C09038=1044.686,246.320,-104.218,171.561,39.501,157.497
C09039=1044.679,246.071,-104.189,171.559,39.498,157.496
C09040=1044.673,245.823,-104.160,171.556,39.496,157.496
C09041=1044.666,245.575,-104.131,171.553,39.493,157.495
C09042=1044.659,245.327,-104.102,171.551,39.491,157.495
C09043=1044.653,245.078,-104.074,171.548,39.489,157.494
C09044=1044.646,244.830,-104.045,171.546,39.486,157.493
C09045=1044.640,244.582,-104.016,171.543,39.484,157.493
C09046=1044.634,244.333,-103.988,171.541,39.481,157.492
C09047=1044.627,244.085,-103.959,171.538,39.479,157.491
C09048=1044.620,243.837,-103.930,171.535,39.476,157.491
C09049=1044.613,243.589,-103.902,171.533,39.474,157.490
C09050=1044.607,243.340,-103.873,171.530,39.472,157.490
C09051=1044.601,243.092,-103.844,171.527,39.469,157.489
C09052=1044.594,242.844,-103.816,171.525,39.467,157.488
C09053=1044.588,242.595,-103.788,171.522,39.464,157.488
C09054=1044.581,242.348,-103.759,171.520,39.462,157.487
C09055=1044.575,242.099,-103.731,171.517,39.459,157.487
C09056=1044.569,241.850,-103.701,171.515,39.457,157.486
C09057=1044.562,241.602,-103.673,171.512,39.455,157.486
C09058=1044.556,241.353,-103.645,171.509,39.452,157.485
C09059=1044.549,241.106,-103.616,171.507,39.449,157.484
C09060=1044.542,240.857,-103.589,171.504,39.447,157.484
C09061=1044.536,240.609,-103.559,171.502,39.445,157.483
C09062=1044.529,240.361,-103.532,171.499,39.443,157.483
C09063=1044.523,240.112,-103.503,171.497,39.440,157.482
C09064=1044.516,239.864,-103.475,171.494,39.437,157.481
C09065=1044.509,239.616,-103.447,171.491,39.435,157.481
C09066=1044.503,239.367,-103.418,171.490,39.433,157.480
C09067=1044.496,239.119,-103.390,171.487,39.431,157.480
C09068=1044.489,238.871,-103.362,171.485,39.428,157.479
C09069=1044.483,238.622,-103.333,171.482,39.426,157.478
C09070=1044.476,238.374,-103.305,171.479,39.423,157.478
C09071=1044.469,238.125,-103.277,171.477,39.421,157.477
C09072=1044.463,237.877,-103.249,171.474,39.419,157.477
C09073=1044.456,237.629,-103.220,171.472,39.416,157.476
C09074=1044.450,237.380,-103.193,171.469,39.414,157.475
C09075=1044.444,237.132,-103.164,171.467,39.411,157.475
C09076=1044.437,236.884,-103.136,171.464,39.409,157.474
C09077=1044.430,236.635,-103.108,171.462,39.407,157.474
C09078=1044.423,236.387,-103.080,171.459,39.404,157.473
C09079=1044.417,236.139,-103.051,171.456,39.402,157.473
C09080=1044.410,235.890,-103.024,171.454,39.400,157.472
C09081=1044.404,235.642,-102.996,171.452,39.397,157.471
C09082=1044.398,235.393,-102.968,171.450,39.394,157.471
C09083=1044.390,235.109,-102.935,171.446,39.392,157.470
C09084=1044.383,234.823,-102.903,171.443,39.389,157.469
C09085=1044.375,234.539,-102.871,171.441,39.387,157.469
C09086=1044.368,234.254,-102.839,171.438,39.384,157.468
C09087=1044.361,234.006,-102.811,171.436,39.381,157.467
C09088=1044.354,233.757,-102.783,171.433,39.378,157.467
C09089=1044.348,233.509,-102.755,171.430,39.376,157.466
C09090=1044.342,233.260,-102.727,171.428,39.374,157.466
C09091=1044.335,233.012,-102.699,171.426,39.372,157.465
C09092=1044.328,232.763,-102.672,171.424,39.369,157.465
C09093=1044.322,232.515,-102.643,171.421,39.366,157.464
C09094=1044.315,232.267,-102.615,171.418,39.364,157.463
C09095=1044.309,232.018,-102.587,171.416,39.362,157.463
C09096=1044.302,231.770,-102.559,171.413,39.360,157.462
C09097=1044.296,231.522,-102.532,171.411,39.357,157.462
C09098=1044.290,231.273,-102.504,171.409,39.354,157.461
C09099=1044.283,231.025,-102.476,171.407,39.352,157.460
C09100=1044.277,230.776,-102.448,171.404,39.350,157.460
C09101=1044.270,230.528,-102.420,171.402,39.347,157.459
C09102=1044.263,230.280,-102.393,171.399,39.345,157.459
C09103=1044.256,230.031,-102.365,171.396,39.342,157.458
C09104=1044.250,229.783,-102.337,171.395,39.340,157.457
C09105=1044.243,229.534,-102.310,171.392,39.338,157.457
C09106=1044.237,229.287,-102.282,171.390,39.335,157.456
C09107=1044.231,229.038,-102.254,171.387,39.333,157.456
C09108=1044.224,228.789,-102.226,171.384,39.330,157.455
C09109=1044.218,228.541,-102.198,171.382,39.328,157.454
C09110=1044.211,228.292,-102.171,171.380,39.325,157.454
C09111=1044.204,228.044,-102.144,171.378,39.323,157.453
C09112=1044.197,227.795,-102.117,171.375,39.321,157.453
C09113=1044.191,227.547,-102.089,171.373,39.319,157.452
C09114=1044.184,227.299,-102.061,171.370,39.316,157.452
C09115=1044.178,227.051,-102.034,171.369,39.314,157.451
C09116=1044.171,226.802,-102.006,171.366,39.312,157.451
C09117=1044.164,226.554,-101.978,171.364,39.309,157.450
C09118=1044.158,226.305,-101.951,171.361,39.306,157.449
C09119=1044.151,226.056,-101.924,171.358,39.304,157.449
C09120=1044.145,225.809,-101.897,171.357,39.302,157.448
C09121=1044.138,225.560,-101.869,171.354,39.299,157.448
C09122=1044.131,225.312,-101.841,171.352,39.297,157.447
C09123=1044.125,225.063,-101.814,171.349,39.295,157.446
C09124=1044.118,224.814,-101.787,171.347,39.292,157.446
C09125=1044.111,224.566,-101.759,171.345,39.290,157.445
C09126=1044.106,224.318,-101.732,171.343,39.287,157.445
C09127=1044.099,224.069,-101.704,171.340,39.285,157.444
C09128=1044.092,223.821,-101.677,171.337,39.283,157.444
C09129=1044.085,223.573,-101.650,171.336,39.280,157.443
C09130=1044.079,223.324,-101.623,171.333,39.277,157.442
C09131=1044.072,223.076,-101.595,171.331,39.275,157.442
C09132=1044.066,222.827,-101.567,171.328,39.273,157.441
C09133=1044.059,222.578,-101.540,171.327,39.271,157.441
C09134=1044.053,222.331,-101.513,171.324,39.268,157.440
C09135=1044.046,222.082,-101.486,171.322,39.266,157.440
C09136=1044.040,221.833,-101.459,171.319,39.263,157.439
C09137=1044.033,221.585,-101.431,171.317,39.261,157.438
C09138=1044.027,221.337,-101.405,171.315,39.258,157.438
C09139=1044.019,221.044,-101.372,171.312,39.255,157.437
C09140=1044.012,220.752,-101.340,171.310,39.253,157.436
C09141=1044.003,220.459,-101.308,171.307,39.250,157.436
C09142=1043.996,220.167,-101.276,171.304,39.247,157.435
C09143=1043.990,219.918,-101.249,171.302,39.244,157.434
C09144=1043.983,219.670,-101.222,171.299,39.242,157.434
C09145=1043.976,219.421,-101.195,171.298,39.240,157.433
C09146=1043.969,219.173,-101.168,171.295,39.237,157.433
C09147=1043.963,218.925,-101.141,171.293,39.235,157.432
C09148=1043.956,218.676,-101.114,171.290,39.233,157.432
C09149=1043.950,218.428,-101.087,171.288,39.230,157.431
C09150=1043.943,218.179,-101.060,171.286,39.228,157.430
C09151=1043.936,217.930,-101.034,171.283,39.225,157.430
C09152=1043.929,217.682,-101.006,171.282,39.223,157.429
C09153=1043.924,217.433,-100.979,171.279,39.221,157.429
C09154=1043.916,217.185,-100.952,171.277,39.218,157.428
C09155=1043.910,216.936,-100.925,171.275,39.216,157.428
C09156=1043.903,216.688,-100.899,171.273,39.213,157.427
C09157=1043.897,216.440,-100.871,171.270,39.211,157.426
C09158=1043.890,216.191,-100.845,171.268,39.208,157.426
C09159=1043.884,215.943,-100.818,171.266,39.206,157.425
C09160=1043.877,215.694,-100.790,171.263,39.204,157.425
C09161=1043.870,215.445,-100.764,171.261,39.201,157.424
C09162=1043.864,215.197,-100.737,171.259,39.199,157.424
C09163=1043.857,214.949,-100.710,171.257,39.196,157.423
C09164=1043.851,214.701,-100.684,171.254,39.194,157.422
C09165=1043.844,214.452,-100.657,171.253,39.191,157.422
C09166=1043.838,214.203,-100.630,171.250,39.189,157.421
C09167=1043.829,213.866,-100.594,171.247,39.186,157.420
C09168=1043.820,213.528,-100.558,171.245,39.182,157.420
C09169=1043.811,213.191,-100.521,171.241,39.179,157.419
C09170=1043.802,212.853,-100.485,171.238,39.176,157.418
C09171=1043.796,212.606,-100.458,171.237,39.173,157.418
C09172=1043.789,212.357,-100.431,171.234,39.171,157.417
C09173=1043.782,212.108,-100.404,171.231,39.168,157.416
C09174=1043.777,211.860,-100.378,171.230,39.166,157.416
C09175=1043.769,211.611,-100.351,171.227,39.163,157.415
C09176=1043.763,211.363,-100.325,171.226,39.161,157.415
C09177=1043.757,211.114,-100.298,171.223,39.159,157.414
C09178=1043.750,210.866,-100.271,171.221,39.156,157.414
C09179=1043.743,210.617,-100.244,171.219,39.153,157.413
C09180=1043.736,210.368,-100.218,171.217,39.151,157.412
C09181=1043.730,210.120,-100.192,171.214,39.149,157.412
C09182=1043.723,209.871,-100.165,171.213,39.146,157.411
C09183=1043.717,209.623,-100.139,171.210,39.144,157.411
C09184=1043.710,209.374,-100.112,171.208,39.141,157.410
C09185=1043.704,209.126,-100.086,171.206,39.139,157.409
C09186=1043.697,208.877,-100.059,171.203,39.137,157.409
C09187=1043.690,208.629,-100.033,171.202,39.134,157.408
C09188=1043.684,208.380,-100.006,171.199,39.132,157.408
C09189=1043.677,208.132,-99.980,171.198,39.129,157.407
C09190=1043.670,207.883,-99.954,171.195,39.127,157.407
C09191=1043.665,207.660,-99.929,171.194,39.125,157.406
C09192=1043.659,207.437,-99.906,171.191,39.122,157.406
C09193=1043.653,207.214,-99.883,171.190,39.120,157.405
C09194=1043.646,206.990,-99.859,171.187,39.118,157.405
C09195=1043.641,206.767,-99.836,171.186,39.116,157.404
C09196=1043.635,206.544,-99.812,171.184,39.114,157.404
C09197=1043.628,206.321,-99.788,171.182,39.111,157.403
C09198=1043.623,206.097,-99.764,171.181,39.110,157.403
C09199=1043.597,205.046,-99.658,170.913,39.008,157.374
C09200=1043.591,204.797,-99.633,170.910,39.006,157.373
C09201=1043.585,204.548,-99.608,170.907,39.004,157.373
C09202=1043.578,204.300,-99.583,170.905,39.003,157.373
C09203=1043.572,204.051,-99.558,170.901,39.001,157.372
C09204=1043.566,203.802,-99.532,170.899,38.999,157.372
C09205=1043.560,203.554,-99.507,170.895,38.998,157.371
C09206=1043.554,203.305,-99.483,170.893,38.996,157.371
C09207=1043.548,203.056,-99.457,170.890,38.994,157.370
C09208=1043.542,202.808,-99.432,170.887,38.993,157.370
C09209=1043.536,202.559,-99.407,170.884,38.991,157.370
C09210=1043.530,202.310,-99.382,170.882,38.989,157.369
C09211=1043.524,202.062,-99.357,170.879,38.987,157.369
C09212=1043.518,201.813,-99.332,170.876,38.986,157.368
C09213=1043.512,201.565,-99.306,170.873,38.984,157.368
C09214=1043.506,201.315,-99.282,170.870,38.982,157.368
C09215=1043.499,201.067,-99.257,170.868,38.981,157.367
C09216=1043.493,200.818,-99.232,170.864,38.979,157.367
C09217=1043.487,200.570,-99.208,170.862,38.978,157.366
C09218=1043.480,200.321,-99.183,170.859,38.976,157.366
C09219=1043.474,200.072,-99.158,170.856,38.975,157.366
C09220=1043.468,199.824,-99.133,170.853,38.973,157.365
C09221=1043.462,199.574,-99.109,170.851,38.972,157.365
C09222=1043.455,199.326,-99.084,170.848,38.970,157.364
C09223=1043.449,199.077,-99.060,170.845,38.968,157.364
C09224=1043.443,198.829,-99.034,170.842,38.967,157.364
C09225=1043.437,198.580,-99.010,170.839,38.966,157.363
C09226=1043.430,198.331,-98.985,170.837,38.964,157.363
C09227=1043.424,198.082,-98.961,170.833,38.962,157.362
C09228=1043.418,197.834,-98.936,170.831,38.961,157.362
C09229=1043.411,197.585,-98.912,170.828,38.960,157.362
C09230=1043.405,197.336,-98.887,170.825,38.958,157.361
C09231=1043.399,197.087,-98.862,170.823,38.956,157.361
C09232=1043.393,196.840,-98.838,170.820,38.954,157.360
C09233=1043.387,196.590,-98.813,170.817,38.953,157.360
C09234=1043.380,196.341,-98.789,170.814,38.952,157.360
C09235=1043.374,196.093,-98.764,170.812,38.950,157.359
C09236=1043.368,195.844,-98.740,170.809,38.949,157.359
C09237=1043.362,195.596,-98.715,170.806,38.947,157.359
C09238=1043.356,195.346,-98.690,170.804,38.945,157.358
C09239=1043.350,195.098,-98.666,170.800,38.944,157.358
C09240=1043.344,194.849,-98.641,170.798,38.943,157.357
C09241=1043.337,194.600,-98.617,170.795,38.941,157.357
C09242=1043.331,194.351,-98.592,170.792,38.939,157.357
C09243=1043.325,194.104,-98.568,170.790,38.938,157.356
C09244=1043.319,193.854,-98.543,170.786,38.937,157.356
C09245=1043.312,193.605,-98.519,170.784,38.935,157.355
C09246=1043.307,193.357,-98.494,170.782,38.934,157.355
C09247=1043.301,193.108,-98.470,170.778,38.932,157.355
C09248=1043.295,192.860,-98.446,170.776,38.930,157.354
C09249=1043.289,192.610,-98.421,170.774,38.929,157.354
C09250=1043.282,192.362,-98.397,170.770,38.928,157.354
C09251=1043.277,192.113,-98.372,170.768,38.926,157.353
C09252=1043.270,191.864,-98.348,170.765,38.925,157.353
C09253=1043.264,191.615,-98.324,170.762,38.923,157.352
C09254=1043.258,191.367,-98.300,170.760,38.921,157.352
C09255=1043.252,191.118,-98.275,170.757,38.920,157.352
C09256=1043.246,190.870,-98.251,170.754,38.919,157.351
C09257=1043.240,190.621,-98.226,170.752,38.917,157.351
C09258=1043.233,190.372,-98.202,170.749,38.916,157.351
C09259=1043.228,190.123,-98.178,170.746,38.914,157.350
C09260=1043.221,189.839,-98.150,170.743,38.912,157.350
C09261=1043.214,189.554,-98.123,170.741,38.911,157.349
C09262=1043.207,189.271,-98.095,170.737,38.909,157.349
C09263=1043.201,188.985,-98.067,170.734,38.907,157.349
C09264=1043.194,188.736,-98.043,170.732,38.906,157.348
C09265=1043.189,188.488,-98.019,170.729,38.905,157.348
C09266=1043.182,188.239,-97.995,170.727,38.903,157.347
C09267=1043.176,187.991,-97.970,170.724,38.902,157.347
C09268=1043.170,187.742,-97.946,170.721,38.900,157.347
C09269=1043.165,187.493,-97.922,170.719,38.899,157.346
C09270=1043.158,187.244,-97.897,170.716,38.897,157.346
C09271=1043.153,186.996,-97.873,170.713,38.895,157.346
C09272=1043.146,186.747,-97.849,170.711,38.894,157.345
C09273=1043.141,186.498,-97.825,170.708,38.893,157.345
C09274=1043.134,186.249,-97.801,170.705,38.892,157.345
C09275=1043.129,186.001,-97.777,170.703,38.890,157.344
C09276=1043.123,185.752,-97.753,170.701,38.888,157.344
C09277=1043.117,185.503,-97.728,170.697,38.887,157.343
C09278=1043.111,185.255,-97.705,170.695,38.885,157.343
C09279=1043.104,185.005,-97.681,170.693,38.884,157.343
C09280=1043.099,184.757,-97.657,170.690,38.882,157.342
C09281=1043.092,184.508,-97.633,170.687,38.881,157.342
C09282=1043.087,184.259,-97.609,170.685,38.880,157.342
C09283=1043.081,184.010,-97.585,170.682,38.878,157.341
C09284=1043.075,183.761,-97.561,170.680,38.877,157.341
C09285=1043.069,183.513,-97.537,170.677,38.875,157.340
C09286=1043.063,183.264,-97.514,170.674,38.874,157.340
C09287=1043.056,183.015,-97.490,170.672,38.873,157.340
C09288=1043.050,182.766,-97.466,170.669,38.872,157.340
C09289=1043.044,182.517,-97.442,170.666,38.870,157.339
C09290=1043.038,182.268,-97.419,170.664,38.869,157.339
C09291=1043.031,182.019,-97.395,170.661,38.868,157.339
C09292=1043.024,181.771,-97.372,170.659,38.866,157.338
C09293=1043.018,181.522,-97.349,170.656,38.865,157.338
C09294=1043.012,181.274,-97.325,170.653,38.864,157.338
C09295=1043.005,181.025,-97.301,170.651,38.863,157.337
C09296=1043.000,180.776,-97.278,170.648,38.861,157.337
C09297=1042.993,180.527,-97.254,170.646,38.860,157.337
C09298=1042.987,180.278,-97.230,170.643,38.859,157.336
C09299=1042.981,180.030,-97.207,170.641,38.858,157.336
C09300=1042.975,179.781,-97.183,170.638,38.856,157.336
C09301=1042.969,179.532,-97.160,170.635,38.855,157.335
C09302=1042.962,179.283,-97.136,170.633,38.854,157.335
C09303=1042.957,179.034,-97.113,170.631,38.853,157.335
C09304=1042.949,178.785,-97.090,170.628,38.851,157.334
C09305=1042.943,178.537,-97.066,170.625,38.850,157.334
C09306=1042.937,178.288,-97.043,170.623,38.849,157.334
C09307=1042.931,178.039,-97.019,170.620,38.848,157.334
C09308=1042.925,177.790,-96.996,170.618,38.846,157.333
C09309=1042.918,177.541,-96.972,170.615,38.845,157.333
C09310=1042.913,177.292,-96.949,170.613,38.844,157.333
C09311=1042.907,177.044,-96.926,170.610,38.843,157.332
C09312=1042.900,176.794,-96.902,170.608,38.841,157.332
C09313=1042.894,176.546,-96.879,170.605,38.840,157.332
C09314=1042.887,176.297,-96.856,170.602,38.839,157.331
C09315=1042.881,176.049,-96.832,170.600,38.838,157.331
C09316=1042.875,175.800,-96.809,170.598,38.837,157.331
C09317=1042.869,175.550,-96.786,170.596,38.835,157.330
C09318=1042.863,175.302,-96.762,170.592,38.834,157.330
C09319=1042.857,175.053,-96.739,170.590,38.833,157.330
C09320=1042.851,174.804,-96.715,170.588,38.832,157.329
C09321=1042.845,174.555,-96.692,170.586,38.831,157.329
C09322=1042.838,174.306,-96.670,170.582,38.829,157.329
C09323=1042.832,174.057,-96.646,170.580,38.828,157.328
C09324=1042.826,173.773,-96.620,170.578,38.827,157.328
C09325=1042.818,173.488,-96.593,170.574,38.825,157.328
C09326=1042.811,173.203,-96.566,170.572,38.823,157.327
C09327=1042.805,172.918,-96.539,170.569,38.822,157.327
C09328=1042.799,172.670,-96.516,170.566,38.821,157.327
C09329=1042.792,172.420,-96.494,170.564,38.820,157.326
C09330=1042.786,172.171,-96.471,170.562,38.818,157.326
C09331=1042.780,171.923,-96.447,170.559,38.817,157.326
C09332=1042.774,171.674,-96.424,170.556,38.816,157.325
C09333=1042.768,171.425,-96.401,170.554,38.815,157.325
C09334=1042.762,171.176,-96.377,170.552,38.814,157.325
C09335=1042.756,170.928,-96.355,170.549,38.812,157.324
C09336=1042.750,170.679,-96.332,170.547,38.811,157.324
C09337=1042.743,170.429,-96.309,170.544,38.810,157.324
C09338=1042.737,170.181,-96.285,170.542,38.809,157.324
C09339=1042.732,169.932,-96.262,170.539,38.808,157.323
C09340=1042.726,169.683,-96.239,170.537,38.806,157.323
C09341=1042.720,169.434,-96.216,170.535,38.805,157.323
C09342=1042.713,169.185,-96.193,170.533,38.804,157.322
C09343=1042.707,168.937,-96.170,170.529,38.803,157.322
C09344=1042.701,168.688,-96.147,170.527,38.801,157.322
C09345=1042.696,168.439,-96.124,170.525,38.800,157.321
C09346=1042.690,168.190,-96.101,170.522,38.799,157.321
C09347=1042.683,167.941,-96.078,170.520,38.797,157.321
C09348=1042.677,167.692,-96.055,170.518,38.796,157.321
C09349=1042.671,167.443,-96.032,170.516,38.795,157.320
C09350=1042.665,167.195,-96.009,170.512,38.794,157.320
C09351=1042.660,166.946,-95.986,170.510,38.792,157.320
C09352=1042.654,166.697,-95.963,170.508,38.791,157.319
C09353=1042.647,166.448,-95.940,170.506,38.790,157.319
C09354=1042.641,166.199,-95.917,170.503,38.789,157.319
C09355=1042.635,165.950,-95.894,170.501,38.788,157.318
C09356=1042.630,165.701,-95.871,170.499,38.787,157.318
C09357=1042.624,165.452,-95.848,170.496,38.785,157.318
C09358=1042.617,165.203,-95.826,170.494,38.784,157.317
C09359=1042.612,164.955,-95.803,170.491,38.783,157.317
C09360=1042.606,164.706,-95.780,170.489,38.782,157.317
C09361=1042.600,164.457,-95.757,170.486,38.781,157.317
C09362=1042.595,164.208,-95.734,170.484,38.779,157.316
C09363=1042.588,163.959,-95.712,170.482,38.778,157.316
C09364=1042.582,163.710,-95.689,170.480,38.777,157.316
C09365=1042.577,163.461,-95.666,170.477,38.775,157.315
C09366=1042.570,163.212,-95.643,170.475,38.774,157.315
C09367=1042.565,162.963,-95.620,170.473,38.773,157.315
C09368=1042.558,162.714,-95.597,170.471,38.772,157.314
C09369=1042.552,162.466,-95.574,170.467,38.770,157.314
C09370=1042.547,162.217,-95.551,170.465,38.769,157.314
C09371=1042.541,161.968,-95.528,170.463,38.768,157.313
C09372=1042.535,161.719,-95.505,170.460,38.767,157.313
C09373=1042.529,161.470,-95.483,170.458,38.766,157.313
C09374=1042.523,161.221,-95.460,170.456,38.765,157.313
C09375=1042.517,160.972,-95.437,170.454,38.763,157.312
C09376=1042.512,160.723,-95.415,170.451,38.762,157.312
C09377=1042.505,160.474,-95.393,170.449,38.761,157.312
C09378=1042.500,160.225,-95.370,170.447,38.760,157.311
C09379=1042.494,159.977,-95.347,170.445,38.758,157.311
C09380=1042.487,159.728,-95.324,170.442,38.757,157.311
C09381=1042.481,159.479,-95.303,170.440,38.756,157.311
C09382=1042.475,159.230,-95.280,170.437,38.755,157.310
C09383=1042.469,158.981,-95.257,170.435,38.754,157.310
C09384=1042.463,158.732,-95.236,170.432,38.753,157.310
C09385=1042.457,158.483,-95.213,170.430,38.752,157.309
C09386=1042.451,158.235,-95.191,170.428,38.751,157.309
C09387=1042.445,157.986,-95.168,170.426,38.749,157.309
C09388=1042.438,157.700,-95.142,170.423,38.748,157.309
C09389=1042.431,157.414,-95.117,170.420,38.747,157.308
C09390=1042.424,157.130,-95.091,170.418,38.746,157.308
C09391=1042.417,156.844,-95.066,170.416,38.745,157.308
C09392=1042.411,156.595,-95.043,170.412,38.744,157.307
C09393=1042.404,156.346,-95.021,170.410,38.743,157.307
C09394=1042.398,156.097,-94.999,170.408,38.742,157.307
C09395=1042.392,155.848,-94.976,170.406,38.741,157.307
C09396=1042.386,155.599,-94.954,170.403,38.739,157.306
C09397=1042.380,155.350,-94.932,170.401,38.738,157.306
C09398=1042.374,155.102,-94.909,170.399,38.737,157.306
C09399=1042.368,154.852,-94.887,170.397,38.736,157.305
C09400=1042.361,154.604,-94.865,170.394,38.735,157.305
C09401=1042.356,154.354,-94.843,170.392,38.734,157.305
C09402=1042.350,154.106,-94.821,170.390,38.733,157.305
C09403=1042.343,153.856,-94.799,170.388,38.732,157.304
C09404=1042.337,153.608,-94.777,170.386,38.731,157.304
C09405=1042.331,153.358,-94.754,170.383,38.730,157.304
C09406=1042.325,153.110,-94.732,170.381,38.729,157.304
C09407=1042.319,152.861,-94.710,170.379,38.728,157.303
C09408=1042.312,152.612,-94.688,170.377,38.726,157.303
C09409=1042.307,152.364,-94.667,170.373,38.725,157.303
C09410=1042.301,152.115,-94.644,170.371,38.724,157.302
C09411=1042.295,151.865,-94.622,170.369,38.724,157.302
C09412=1042.288,151.617,-94.600,170.367,38.723,157.302
C09413=1042.282,151.368,-94.578,170.364,38.721,157.302
C09414=1042.277,151.118,-94.556,170.362,38.720,157.302
C09415=1042.270,150.870,-94.534,170.360,38.719,157.301
C09416=1042.264,150.620,-94.512,170.358,38.718,157.301
C09417=1042.258,150.372,-94.490,170.355,38.717,157.301
C09418=1042.252,150.123,-94.468,170.353,38.716,157.300
C09419=1042.246,149.873,-94.446,170.351,38.715,157.300
C09420=1042.240,149.624,-94.423,170.349,38.714,157.300
C09421=1042.234,149.376,-94.402,170.347,38.713,157.300
C09422=1042.228,149.127,-94.380,170.344,38.712,157.299
C09423=1042.222,148.878,-94.358,170.342,38.711,157.299
C09424=1042.215,148.629,-94.336,170.340,38.710,157.299
C09425=1042.209,148.380,-94.315,170.338,38.709,157.299
C09426=1042.203,148.131,-94.292,170.335,38.708,157.298
C09427=1042.197,147.882,-94.270,170.333,38.707,157.298
C09428=1042.191,147.632,-94.249,170.331,38.706,157.298
C09429=1042.186,147.384,-94.227,170.329,38.705,157.298
C09430=1042.179,147.135,-94.205,170.326,38.703,157.297
C09431=1042.173,146.886,-94.183,170.324,38.703,157.297
C09432=1042.167,146.637,-94.162,170.322,38.702,157.297
C09433=1042.161,146.388,-94.140,170.320,38.701,157.297
C09434=1042.154,146.138,-94.118,170.318,38.699,157.296
C09435=1042.148,145.890,-94.096,170.315,38.699,157.296
C09436=1042.142,145.641,-94.075,170.313,38.698,157.296
C09437=1042.136,145.392,-94.053,170.311,38.697,157.296
C09438=1042.130,145.143,-94.032,170.309,38.696,157.295
C09439=1042.124,144.894,-94.010,170.307,38.695,157.295
C09440=1042.118,144.645,-93.988,170.304,38.694,157.295
C09441=1042.111,144.396,-93.966,170.302,38.693,157.295
C09442=1042.106,144.147,-93.945,170.300,38.692,157.294
C09443=1042.099,143.899,-93.924,170.298,38.691,157.294
C09444=1042.093,143.649,-93.902,170.296,38.690,157.294
C09445=1042.087,143.400,-93.880,170.293,38.689,157.294
C09446=1042.080,143.151,-93.859,170.291,38.688,157.293
C09447=1042.074,142.902,-93.837,170.289,38.687,157.293
C09448=1042.069,142.653,-93.816,170.287,38.686,157.293
C09449=1042.062,142.404,-93.794,170.284,38.685,157.293
C09450=1042.056,142.155,-93.773,170.282,38.684,157.292
C09451=1042.050,141.906,-93.751,170.280,38.683,157.292
C09452=1042.044,141.621,-93.726,170.278,38.682,157.292
C09453=1042.036,141.335,-93.701,170.275,38.681,157.292
C09454=1042.029,141.049,-93.677,170.272,38.680,157.291
C09455=1042.022,140.764,-93.652,170.270,38.679,157.291
C09456=1042.017,140.515,-93.630,170.268,38.678,157.291
C09457=1042.010,140.266,-93.609,170.266,38.677,157.291
C09458=1042.004,140.017,-93.587,170.263,38.676,157.290
C09459=1041.997,139.768,-93.566,170.261,38.675,157.290
C09460=1041.992,139.519,-93.545,170.259,38.674,157.290
C09461=1041.986,139.270,-93.523,170.257,38.673,157.290
C09462=1041.980,139.021,-93.502,170.255,38.672,157.289
C09463=1041.974,138.771,-93.481,170.252,38.671,157.289
C09464=1041.968,138.523,-93.459,170.250,38.670,157.289
C09465=1041.961,138.274,-93.438,170.248,38.669,157.289
C09466=1041.955,138.024,-93.417,170.246,38.668,157.288
C09467=1041.949,137.775,-93.395,170.244,38.667,157.288
C09468=1041.943,137.527,-93.374,170.241,38.666,157.288
C09469=1041.936,137.278,-93.353,170.239,38.665,157.288
C09470=1041.930,137.029,-93.331,170.237,38.664,157.287
C09471=1041.924,136.779,-93.310,170.235,38.664,157.287
C09472=1041.918,136.531,-93.289,170.233,38.663,157.287
C09473=1041.912,136.281,-93.268,170.230,38.661,157.287
C09474=1041.906,136.032,-93.246,170.229,38.661,157.287
C09475=1041.900,135.784,-93.225,170.227,38.660,157.286
C09476=1041.894,135.534,-93.205,170.225,38.659,157.286
C09477=1041.887,135.285,-93.183,170.223,38.658,157.286
C09478=1041.882,135.036,-93.162,170.220,38.657,157.286
C09479=1041.875,134.788,-93.141,170.218,38.656,157.285
C09480=1041.869,134.538,-93.120,170.216,38.655,157.285
C09481=1041.864,134.289,-93.098,170.214,38.654,157.285
C09482=1041.857,134.040,-93.077,170.211,38.653,157.285
C09483=1041.851,133.791,-93.056,170.209,38.652,157.284
C09484=1041.845,133.542,-93.035,170.207,38.651,157.284
C09485=1041.838,133.293,-93.014,170.205,38.651,157.284
C09486=1041.832,133.044,-92.993,170.203,38.650,157.284
C09487=1041.827,132.795,-92.971,170.200,38.648,157.283
C09488=1041.820,132.546,-92.951,170.198,38.648,157.283
C09489=1041.814,132.297,-92.929,170.196,38.647,157.283
C09490=1041.808,132.048,-92.908,170.194,38.646,157.283
C09491=1041.802,131.799,-92.888,170.193,38.645,157.283
C09492=1041.796,131.550,-92.866,170.191,38.644,157.282
C09493=1041.790,131.301,-92.845,170.188,38.643,157.282
C09494=1041.783,131.051,-92.825,170.186,38.642,157.282
C09495=1041.778,130.803,-92.803,170.184,38.641,157.282
C09496=1041.771,130.553,-92.783,170.182,38.641,157.281
C09497=1041.764,130.305,-92.762,170.180,38.640,157.281
C09498=1041.759,130.055,-92.741,170.177,38.639,157.281
C09499=1041.752,129.807,-92.720,170.175,38.638,157.281
C09500=1041.746,129.557,-92.700,170.173,38.637,157.281
C09501=1041.740,129.309,-92.679,170.171,38.636,157.280
C09502=1041.733,129.059,-92.658,170.169,38.636,157.280
C09503=1041.727,128.810,-92.637,170.166,38.635,157.280
C09504=1041.721,128.561,-92.617,170.164,38.634,157.280
C09505=1041.714,128.312,-92.596,170.162,38.633,157.279
C09506=1041.708,128.063,-92.575,170.160,38.632,157.279
C09507=1041.702,127.814,-92.554,170.158,38.631,157.279
C09508=1041.696,127.565,-92.534,170.157,38.631,157.279
C09509=1041.690,127.316,-92.513,170.154,38.629,157.279
C09510=1041.683,127.067,-92.492,170.152,38.629,157.278
C09511=1041.677,126.818,-92.471,170.150,38.628,157.278
C09512=1041.671,126.569,-92.451,170.148,38.627,157.278
C09513=1041.665,126.319,-92.430,170.146,38.626,157.278
C09514=1041.658,126.071,-92.410,170.143,38.626,157.278
C09515=1041.653,125.821,-92.389,170.141,38.625,157.277
C09516=1041.646,125.536,-92.365,170.139,38.623,157.277
C09517=1041.638,125.249,-92.341,170.137,38.623,157.277
C09518=1041.631,124.964,-92.317,170.134,38.622,157.277
C09519=1041.624,124.678,-92.294,170.131,38.621,157.276
C09520=1041.617,124.429,-92.273,170.129,38.620,157.276
C09521=1041.611,124.179,-92.252,170.127,38.619,157.276
C09522=1041.605,123.931,-92.233,170.126,38.618,157.276
C09523=1041.599,123.682,-92.211,170.124,38.617,157.276
C09524=1041.593,123.433,-92.191,170.122,38.617,157.275
C09525=1041.587,123.183,-92.171,170.119,38.616,157.275
C09526=1041.580,122.935,-92.150,170.117,38.615,157.275
C09527=1041.574,122.685,-92.130,170.115,38.614,157.275
C09528=1041.569,122.436,-92.109,170.113,38.613,157.274
C09529=1041.562,122.187,-92.088,170.111,38.612,157.274
C09530=1041.556,121.938,-92.068,170.108,38.611,157.274
C09531=1041.550,121.689,-92.047,170.106,38.611,157.274
C09532=1041.544,121.440,-92.027,170.105,38.609,157.274
C09533=1041.537,121.191,-92.006,170.103,38.609,157.273
C09534=1041.532,120.942,-91.986,170.101,38.608,157.273
C09535=1041.525,120.692,-91.965,170.098,38.607,157.273
C09536=1041.519,120.443,-91.945,170.096,38.606,157.273
C09537=1041.514,120.195,-91.924,170.094,38.605,157.273
C09538=1041.507,119.945,-91.904,170.092,38.604,157.272
C09539=1041.501,119.697,-91.884,170.090,38.604,157.272
C09540=1041.494,119.447,-91.863,170.089,38.603,157.272
C09541=1041.489,119.199,-91.842,170.086,38.601,157.272
C09542=1041.482,118.949,-91.822,170.084,38.601,157.271
C09543=1041.476,118.700,-91.802,170.082,38.600,157.271
C09544=1041.470,118.450,-91.781,170.080,38.599,157.271
C09545=1041.464,118.202,-91.761,170.078,38.598,157.271
C09546=1041.458,117.953,-91.741,170.075,38.598,157.271
C09547=1041.451,117.704,-91.720,170.073,38.596,157.270
C09548=1041.446,117.455,-91.699,170.072,38.596,157.270
C09549=1041.440,117.205,-91.679,170.070,38.595,157.270
C09550=1041.434,116.956,-91.659,170.068,38.594,157.270
C09551=1041.428,116.707,-91.639,170.065,38.593,157.269
C09552=1041.422,116.458,-91.618,170.063,38.592,157.269
C09553=1041.416,116.209,-91.598,170.061,38.591,157.269
C09554=1041.410,115.960,-91.578,170.059,38.590,157.269
C09555=1041.404,115.710,-91.557,170.058,38.590,157.269
C09556=1041.398,115.462,-91.537,170.055,38.589,157.268
C09557=1041.391,115.213,-91.516,170.053,38.588,157.268
C09558=1041.385,114.964,-91.496,170.051,38.587,157.268
C09559=1041.380,114.715,-91.476,170.049,38.586,157.268
C09560=1041.373,114.465,-91.456,170.047,38.585,157.267
C09561=1041.367,114.216,-91.436,170.046,38.584,157.267
C09562=1041.362,113.967,-91.415,170.043,38.583,157.267
C09563=1041.355,113.718,-91.395,170.041,38.582,157.267
C09564=1041.349,113.469,-91.375,170.039,38.582,157.267
C09565=1041.343,113.220,-91.355,170.037,38.581,157.266
C09566=1041.337,112.971,-91.335,170.035,38.580,157.266
C09567=1041.331,112.722,-91.315,170.032,38.579,157.266
C09568=1041.325,112.473,-91.295,170.031,38.578,157.266
C09569=1041.318,112.224,-91.274,170.029,38.577,157.266
C09570=1041.312,111.975,-91.254,170.027,38.577,157.265
C09571=1041.306,111.725,-91.235,170.025,38.576,157.265
C09572=1041.300,111.476,-91.215,170.023,38.575,157.265
C09573=1041.294,111.227,-91.195,170.020,38.574,157.265
C09574=1041.287,110.977,-91.174,170.018,38.573,157.265
C09575=1041.281,110.729,-91.154,170.017,38.573,157.264
C09576=1041.275,110.480,-91.135,170.015,38.572,157.264
C09577=1041.269,110.230,-91.114,170.013,38.571,157.264
C09578=1041.263,109.981,-91.095,170.011,38.571,157.264
C09579=1041.257,109.732,-91.075,170.008,38.569,157.264
C09580=1041.249,109.421,-91.050,170.006,38.568,157.263
C09581=1041.241,109.110,-91.026,170.003,38.568,157.263
C09582=1041.233,108.799,-91.001,170.001,38.567,157.263
C09583=1041.226,108.489,-90.976,169.999,38.565,157.263
C09584=1041.220,108.252,-90.957,169.996,38.565,157.262
C09585=1041.213,108.015,-90.938,169.994,38.564,157.262
C09586=1041.208,107.779,-90.919,169.992,38.563,157.262
C09587=1041.202,107.542,-90.901,169.991,38.563,157.262
C09588=1041.196,107.305,-90.882,169.989,38.562,157.262
C09589=1041.189,107.068,-90.863,169.987,38.561,157.261
C09590=1041.184,106.832,-90.844,169.984,38.561,157.261
C09591=1041.178,106.595,-90.826,169.983,38.560,157.261
C09592=1041.172,106.346,-90.806,169.981,38.559,157.261
C09593=1041.166,106.097,-90.786,169.979,38.558,157.261
C09594=1041.160,105.848,-90.766,169.977,38.558,157.261
C09595=1041.153,105.598,-90.746,169.975,38.557,157.260
C09596=1041.147,105.349,-90.726,169.973,38.556,157.260
C09597=1041.141,105.101,-90.707,169.971,38.555,157.260
C09598=1041.134,104.851,-90.688,169.969,38.554,157.260
C09599=1041.128,104.602,-90.668,169.967,38.554,157.260
C09600=1041.122,104.353,-90.648,169.965,38.553,157.259
C09601=1041.117,104.104,-90.628,169.963,38.552,157.259
C09602=1041.111,103.855,-90.608,169.960,38.551,157.259
C09603=1041.104,103.605,-90.589,169.959,38.550,157.259
C09604=1041.098,103.356,-90.569,169.957,38.550,157.259
C09605=1041.092,103.107,-90.549,169.955,38.549,157.258
C09606=1041.086,102.858,-90.530,169.953,38.548,157.258
C09607=1041.079,102.608,-90.510,169.951,38.547,157.258
C09608=1041.073,102.359,-90.491,169.948,38.546,157.258
C09609=1041.067,102.110,-90.471,169.947,38.546,157.258
C09610=1041.061,101.862,-90.451,169.945,38.545,157.257
C09611=1041.055,101.612,-90.432,169.943,38.544,157.257
C09612=1041.049,101.363,-90.412,169.941,38.543,157.257
C09613=1041.042,101.114,-90.393,169.939,38.543,157.257
C09614=1041.036,100.865,-90.373,169.936,38.541,157.257
C09615=1041.030,100.615,-90.354,169.935,38.541,157.256
C09616=1041.024,100.366,-90.334,169.933,38.540,157.256
C09617=1041.017,100.117,-90.315,169.931,38.539,157.256
C09618=1041.011,99.868,-90.295,169.929,38.539,157.256
C09619=1041.005,99.619,-90.276,169.927,38.538,157.256
C09620=1040.999,99.370,-90.256,169.924,38.537,157.255
C09621=1040.993,99.120,-90.237,169.923,38.536,157.255
C09622=1040.986,98.871,-90.217,169.921,38.536,157.255
C09623=1040.980,98.622,-90.198,169.919,38.535,157.255
C09624=1040.974,98.373,-90.179,169.917,38.534,157.255
C09625=1040.968,98.124,-90.160,169.915,38.534,157.255
C09626=1040.961,97.875,-90.141,169.913,38.533,157.254
C09627=1040.955,97.625,-90.121,169.911,38.532,157.254
C09628=1040.948,97.376,-90.102,169.909,38.531,157.254
C09629=1040.943,97.127,-90.083,169.907,38.531,157.254
C09630=1040.936,96.878,-90.063,169.905,38.530,157.254
C09631=1040.930,96.629,-90.044,169.903,38.529,157.253
C09632=1040.924,96.380,-90.025,169.901,38.529,157.253
C09633=1040.917,96.130,-90.005,169.899,38.527,157.253
C09634=1040.912,95.881,-89.986,169.897,38.527,157.253
C09635=1040.905,95.632,-89.967,169.895,38.526,157.253
C09636=1040.899,95.383,-89.947,169.893,38.525,157.252
C09637=1040.893,95.134,-89.929,169.891,38.525,157.252
C09638=1040.887,94.884,-89.909,169.889,38.524,157.252
C09639=1040.880,94.636,-89.890,169.887,38.523,157.252
C09640=1040.875,94.386,-89.871,169.885,38.522,157.252
C09641=1040.868,94.136,-89.852,169.883,38.522,157.252
C09642=1040.862,93.888,-89.832,169.881,38.521,157.251
C09643=1040.855,93.639,-89.813,169.879,38.520,157.251
C09644=1040.848,93.352,-89.791,169.877,38.520,157.251
C09645=1040.841,93.066,-89.769,169.874,38.518,157.251
C09646=1040.835,92.781,-89.747,169.872,38.518,157.251
C09647=1040.827,92.495,-89.725,169.870,38.517,157.250
C09648=1040.821,92.246,-89.706,169.868,38.516,157.250
C09649=1040.815,91.996,-89.687,169.866,38.515,157.250
C09650=1040.808,91.746,-89.668,169.864,38.515,157.250
C09651=1040.802,91.498,-89.648,169.863,38.514,157.250
C09652=1040.796,91.249,-89.629,169.860,38.513,157.249
C09653=1040.790,90.999,-89.610,169.858,38.512,157.249
C09654=1040.784,90.750,-89.592,169.856,38.512,157.249
C09655=1040.778,90.501,-89.572,169.854,38.511,157.249
C09656=1040.772,90.251,-89.554,169.853,38.510,157.249
C09657=1040.766,90.003,-89.534,169.851,38.509,157.248
C09658=1040.759,89.754,-89.515,169.848,38.508,157.248
C09659=1040.753,89.504,-89.496,169.846,38.508,157.248
C09660=1040.746,89.255,-89.478,169.844,38.507,157.248
C09661=1040.741,89.006,-89.458,169.842,38.507,157.248
C09662=1040.734,88.757,-89.440,169.841,38.506,157.247
C09663=1040.728,88.508,-89.421,169.839,38.505,157.247
C09664=1040.721,88.258,-89.402,169.837,38.504,157.247
C09665=1040.715,88.008,-89.383,169.834,38.504,157.247
C09666=1040.709,87.759,-89.364,169.832,38.503,157.247
C09667=1040.702,87.510,-89.346,169.830,38.502,157.247
C09668=1040.696,87.261,-89.327,169.829,38.502,157.246
C09669=1040.690,87.012,-89.308,169.827,38.501,157.246
C09670=1040.684,86.762,-89.289,169.825,38.501,157.246
C09671=1040.677,86.513,-89.270,169.822,38.499,157.246
C09672=1040.671,86.264,-89.252,169.820,38.499,157.246
C09673=1040.664,86.015,-89.233,169.818,38.498,157.246
C09674=1040.659,85.766,-89.214,169.817,38.498,157.245
C09675=1040.652,85.516,-89.195,169.815,38.497,157.245
C09676=1040.646,85.267,-89.177,169.813,38.496,157.245
C09677=1040.639,85.018,-89.158,169.811,38.496,157.245
C09678=1040.633,84.769,-89.139,169.808,38.495,157.245
C09679=1040.627,84.520,-89.120,169.807,38.494,157.245
C09680=1040.621,84.271,-89.101,169.805,38.493,157.244
C09681=1040.615,84.021,-89.083,169.803,38.493,157.244
C09682=1040.608,83.772,-89.064,169.801,38.492,157.244
C09683=1040.602,83.523,-89.045,169.799,38.492,157.244
C09684=1040.596,83.274,-89.026,169.797,38.491,157.244
C09685=1040.590,83.025,-89.008,169.795,38.490,157.243
C09686=1040.583,82.775,-88.990,169.793,38.489,157.243
C09687=1040.577,82.526,-88.971,169.791,38.488,157.243
C09688=1040.571,82.276,-88.952,169.789,38.488,157.243
C09689=1040.565,82.027,-88.933,169.787,38.487,157.243
C09690=1040.558,81.778,-88.914,169.786,38.487,157.243
C09691=1040.552,81.529,-88.896,169.783,38.485,157.242
C09692=1040.546,81.281,-88.878,169.781,38.485,157.242
C09693=1040.540,81.031,-88.860,169.779,38.484,157.242
C09694=1040.534,80.781,-88.840,169.777,38.484,157.242
C09695=1040.528,80.532,-88.822,169.775,38.483,157.242
C09696=1040.522,80.283,-88.803,169.774,38.482,157.242
C09697=1040.515,80.034,-88.784,169.772,38.482,157.241
C09698=1040.509,79.785,-88.766,169.769,38.480,157.241
C09699=1040.503,79.535,-88.747,169.767,38.480,157.241
C09700=1040.497,79.286,-88.729,169.765,38.479,157.241
C09701=1040.490,79.037,-88.710,169.764,38.479,157.241
C09702=1040.485,78.788,-88.692,169.762,38.478,157.240
C09703=1040.479,78.538,-88.674,169.760,38.477,157.240
C09704=1040.472,78.289,-88.655,169.758,38.477,157.240
C09705=1040.466,78.040,-88.636,169.755,38.476,157.240
C09706=1040.459,77.791,-88.618,169.754,38.475,157.240
C09707=1040.453,77.541,-88.600,169.752,38.474,157.240
C09708=1040.446,77.255,-88.578,169.750,38.474,157.239
C09709=1040.439,76.969,-88.557,169.748,38.473,157.239
C09710=1040.432,76.683,-88.536,169.746,38.472,157.239
C09711=1040.424,76.397,-88.514,169.742,38.472,157.239
C09712=1040.418,76.147,-88.496,169.741,38.470,157.239
C09713=1040.413,75.899,-88.478,169.739,38.470,157.238
C09714=1040.406,75.649,-88.461,169.737,38.469,157.238
C09715=1040.399,75.400,-88.442,169.735,38.469,157.238
C09716=1040.393,75.151,-88.423,169.733,38.468,157.238
C09717=1040.387,74.901,-88.406,169.731,38.468,157.238
C09718=1040.380,74.652,-88.387,169.729,38.466,157.238
C09719=1040.374,74.403,-88.369,169.727,38.466,157.237
C09720=1040.368,74.153,-88.350,169.725,38.465,157.237
C09721=1040.362,73.905,-88.332,169.723,38.465,157.237
C09722=1040.356,73.655,-88.314,169.721,38.464,157.237
C09723=1040.349,73.406,-88.295,169.719,38.463,157.237
C09724=1040.343,73.156,-88.277,169.718,38.463,157.237
C09725=1040.337,72.907,-88.259,169.715,38.462,157.236
C09726=1040.330,72.658,-88.241,169.713,38.461,157.236
C09727=1040.324,72.410,-88.223,169.711,38.461,157.236
C09728=1040.318,72.160,-88.205,169.709,38.460,157.236
C09729=1040.312,71.911,-88.187,169.708,38.459,157.236
C09730=1040.305,71.662,-88.168,169.706,38.459,157.236
C09731=1040.299,71.412,-88.150,169.704,38.458,157.235
C09732=1040.293,71.163,-88.132,169.702,38.458,157.235
C09733=1040.287,70.914,-88.114,169.699,38.457,157.235
C09734=1040.280,70.664,-88.096,169.697,38.456,157.235
C09735=1040.274,70.415,-88.078,169.696,38.455,157.235
C09736=1040.268,70.165,-88.060,169.694,38.455,157.235
C09737=1040.262,69.917,-88.042,169.692,38.454,157.234
C09738=1040.256,69.667,-88.024,169.690,38.454,157.234
C09739=1040.249,69.418,-88.005,169.687,38.453,157.234
C09740=1040.243,69.168,-87.987,169.686,38.452,157.234
C09741=1040.236,68.919,-87.969,169.684,38.451,157.234
C09742=1040.230,68.670,-87.951,169.682,38.451,157.234
C09743=1040.224,68.421,-87.934,169.680,38.450,157.233
C09744=1040.218,68.172,-87.915,169.678,38.450,157.233
C09745=1040.211,67.922,-87.898,169.676,38.449,157.233
C09746=1040.205,67.672,-87.880,169.675,38.448,157.233
C09747=1040.199,67.424,-87.861,169.672,38.447,157.233
C09748=1040.193,67.174,-87.843,169.670,38.447,157.233
C09749=1040.186,66.925,-87.826,169.668,38.446,157.232
C09750=1040.180,66.676,-87.807,169.666,38.446,157.232
C09751=1040.174,66.427,-87.790,169.664,38.445,157.232
C09752=1040.167,66.177,-87.773,169.663,38.444,157.232
C09753=1040.161,65.928,-87.754,169.661,38.444,157.232
C09754=1040.155,65.678,-87.736,169.658,38.443,157.232
C09755=1040.149,65.430,-87.719,169.656,38.443,157.231
C09756=1040.142,65.181,-87.700,169.654,38.442,157.231
C09757=1040.136,64.931,-87.682,169.652,38.441,157.231
C09758=1040.129,64.681,-87.665,169.651,38.441,157.231
C09759=1040.124,64.432,-87.647,169.649,38.440,157.231
C09760=1040.117,64.183,-87.629,169.647,38.439,157.231
C09761=1040.110,63.934,-87.612,169.644,38.439,157.230
C09762=1040.104,63.684,-87.594,169.642,38.438,157.230
C09763=1040.098,63.435,-87.577,169.640,38.438,157.230
C09764=1040.092,63.186,-87.559,169.639,38.437,157.230
C09765=1040.085,62.936,-87.541,169.637,38.436,157.230
C09766=1040.079,62.687,-87.523,169.635,38.436,157.230
C09767=1040.072,62.438,-87.506,169.633,38.435,157.230
C09768=1040.065,62.189,-87.488,169.631,38.435,157.229
C09769=1040.059,61.939,-87.470,169.629,38.434,157.229
C09770=1040.052,61.690,-87.453,169.626,38.434,157.229
C09771=1040.047,61.441,-87.436,169.624,38.433,157.229
C09772=1040.039,61.154,-87.415,169.622,38.433,157.229
C09773=1040.032,60.868,-87.396,169.620,38.432,157.229
C09774=1040.024,60.582,-87.376,169.618,38.432,157.229
C09775=1040.017,60.296,-87.356,169.616,38.431,157.228
C09776=1040.011,60.047,-87.337,169.614,38.431,157.228
C09777=1040.004,59.797,-87.320,169.612,38.430,157.228
C09778=1039.998,59.547,-87.302,169.609,38.429,157.228
C09779=1039.991,59.299,-87.285,169.607,38.428,157.228
C09780=1039.985,59.049,-87.267,169.606,38.428,157.228
C09781=1039.979,58.800,-87.249,169.604,38.427,157.227
C09782=1039.972,58.551,-87.232,169.602,38.427,157.227
C09783=1039.965,58.301,-87.215,169.600,38.426,157.227
C09784=1039.959,58.052,-87.197,169.598,38.426,157.227
C09785=1039.953,57.803,-87.180,169.595,38.425,157.227
C09786=1039.947,57.553,-87.162,169.593,38.424,157.227
C09787=1039.940,57.304,-87.145,169.592,38.424,157.227
C09788=1039.934,57.055,-87.128,169.590,38.423,157.226
C09789=1039.928,56.805,-87.110,169.588,38.423,157.226
C09790=1039.921,56.556,-87.093,169.586,38.422,157.226
C09791=1039.915,56.307,-87.076,169.584,38.422,157.226
C09792=1039.908,56.057,-87.058,169.582,38.421,157.226
C09793=1039.902,55.809,-87.041,169.580,38.421,157.226
C09794=1039.896,55.559,-87.023,169.578,38.420,157.226
C09795=1039.889,55.310,-87.006,169.576,38.420,157.225
C09796=1039.883,55.060,-86.989,169.574,38.419,157.225
C09797=1039.877,54.810,-86.971,169.572,38.418,157.225
C09798=1039.871,54.562,-86.954,169.570,38.418,157.225
C09799=1039.864,54.312,-86.937,169.568,38.417,157.225
C09800=1039.858,54.063,-86.919,169.566,38.417,157.225
C09801=1039.852,53.814,-86.902,169.565,38.416,157.225
C09802=1039.845,53.564,-86.885,169.562,38.415,157.224
C09803=1039.839,53.315,-86.867,169.560,38.415,157.224
C09804=1039.832,53.066,-86.850,169.558,38.414,157.224
C09805=1039.827,52.816,-86.833,169.556,38.413,157.224
C09806=1039.820,52.567,-86.816,169.554,38.413,157.224
C09807=1039.813,52.317,-86.798,169.552,38.412,157.224
C09808=1039.808,52.068,-86.781,169.551,38.412,157.223
C09809=1039.801,51.819,-86.763,169.549,38.411,157.223
C09810=1039.795,51.570,-86.746,169.546,38.411,157.223
C09811=1039.789,51.320,-86.729,169.544,38.410,157.223
C09812=1039.783,51.071,-86.712,169.542,38.410,157.223
C09813=1039.776,50.822,-86.695,169.540,38.409,157.223
C09814=1039.770,50.573,-86.677,169.539,38.409,157.223
C09815=1039.764,50.323,-86.660,169.537,38.407,157.222
C09816=1039.758,50.074,-86.644,169.535,38.407,157.222
C09817=1039.751,49.824,-86.626,169.532,38.406,157.222
C09818=1039.745,49.575,-86.609,169.530,38.406,157.222
C09819=1039.738,49.326,-86.592,169.528,38.405,157.222
C09820=1039.733,49.077,-86.574,169.526,38.405,157.222
C09821=1039.726,48.827,-86.557,169.525,38.404,157.221
C09822=1039.720,48.578,-86.540,169.523,38.403,157.221
C09823=1039.714,48.328,-86.522,169.521,38.403,157.221
C09824=1039.708,48.079,-86.506,169.519,38.402,157.221
C09825=1039.701,47.830,-86.489,169.516,38.401,157.221
C09826=1039.696,47.581,-86.471,169.514,38.401,157.221
C09827=1039.689,47.331,-86.454,169.512,38.400,157.220
C09828=1039.683,47.082,-86.438,169.511,38.400,157.220
C09829=1039.676,46.832,-86.420,169.509,38.399,157.220
C09830=1039.670,46.583,-86.403,169.507,38.398,157.220
C09831=1039.664,46.333,-86.386,169.505,38.398,157.220
C09832=1039.658,46.085,-86.369,169.503,38.397,157.220
C09833=1039.652,45.835,-86.352,169.500,38.397,157.220
C09834=1039.646,45.585,-86.335,169.499,38.396,157.219
C09835=1039.639,45.337,-86.318,169.497,38.395,157.219
C09836=1039.632,45.049,-86.298,169.495,38.395,157.219
C09837=1039.625,44.764,-86.278,169.492,38.394,157.219
C09838=1039.618,44.477,-86.259,169.490,38.393,157.219
C09839=1039.611,44.190,-86.240,169.488,38.392,157.218
C09840=1039.605,43.941,-86.223,169.485,38.392,157.218
C09841=1039.598,43.692,-86.205,169.484,38.391,157.218
C09842=1039.593,43.442,-86.188,169.482,38.391,157.218
C09843=1039.587,43.193,-86.172,169.480,38.390,157.218
C09844=1039.580,42.943,-86.155,169.478,38.390,157.218
C09845=1039.574,42.694,-86.138,169.476,38.389,157.218
C09846=1039.567,42.444,-86.121,169.474,38.388,157.217
C09847=1039.561,42.196,-86.104,169.472,38.388,157.217
C09848=1039.554,41.946,-86.088,169.469,38.387,157.217
C09849=1039.548,41.697,-86.071,169.468,38.387,157.217
C09850=1039.542,41.447,-86.054,169.466,38.386,157.217
C09851=1039.535,41.198,-86.037,169.464,38.386,157.217
C09852=1039.529,40.949,-86.021,169.462,38.385,157.217
C09853=1039.522,40.699,-86.004,169.460,38.385,157.216
C09854=1039.517,40.450,-85.987,169.458,38.384,157.216
C09855=1039.511,40.200,-85.970,169.456,38.384,157.216
C09856=1039.504,39.951,-85.953,169.454,38.383,157.216
C09857=1039.499,39.701,-85.937,169.451,38.382,157.216
C09858=1039.492,39.452,-85.920,169.450,38.381,157.216
C09859=1039.486,39.203,-85.903,169.448,38.381,157.215
C09860=1039.479,38.954,-85.886,169.446,38.380,157.215
C09861=1039.473,38.704,-85.870,169.444,38.380,157.215
C09862=1039.467,38.455,-85.853,169.442,38.379,157.215
C09863=1039.461,38.206,-85.836,169.440,38.379,157.215
C09864=1039.454,37.956,-85.820,169.437,38.378,157.215
C09865=1039.448,37.706,-85.804,169.435,38.377,157.215
C09866=1039.442,37.458,-85.787,169.433,38.377,157.214
C09867=1039.435,37.208,-85.770,169.432,38.376,157.214
C09868=1039.429,36.958,-85.754,169.430,38.376,157.214
C09869=1039.422,36.710,-85.737,169.428,38.376,157.214
C09870=1039.416,36.460,-85.721,169.426,38.375,157.214
C09871=1039.410,36.210,-85.704,169.424,38.375,157.214
C09872=1039.403,35.960,-85.688,169.422,38.374,157.214
C09873=1039.397,35.712,-85.671,169.420,38.374,157.214
C09874=1039.391,35.462,-85.655,169.417,38.373,157.213
C09875=1039.384,35.213,-85.639,169.415,38.373,157.213
C09876=1039.378,34.963,-85.622,169.413,38.372,157.213
C09877=1039.372,34.715,-85.605,169.411,38.372,157.213
C09878=1039.365,34.464,-85.589,169.410,38.371,157.213
C09879=1039.359,34.215,-85.572,169.408,38.370,157.213
C09880=1039.352,33.966,-85.557,169.406,38.370,157.213
C09881=1039.346,33.717,-85.539,169.404,38.370,157.212
C09882=1039.340,33.467,-85.523,169.402,38.369,157.212
C09883=1039.334,33.218,-85.507,169.399,38.369,157.212
C09884=1039.328,32.969,-85.491,169.397,38.368,157.212
C09885=1039.320,32.719,-85.475,169.395,38.368,157.212
C09886=1039.315,32.470,-85.458,169.393,38.367,157.212
C09887=1039.308,32.221,-85.441,169.391,38.367,157.212
C09888=1039.302,31.971,-85.425,169.389,38.366,157.211
C09889=1039.295,31.722,-85.409,169.387,38.366,157.211
C09890=1039.289,31.472,-85.393,169.385,38.365,157.211
C09891=1039.283,31.223,-85.377,169.383,38.364,157.211
C09892=1039.277,30.973,-85.360,169.381,38.364,157.211
C09893=1039.271,30.724,-85.344,169.379,38.363,157.211
C09894=1039.264,30.475,-85.327,169.377,38.363,157.211
C09895=1039.258,30.226,-85.311,169.375,38.363,157.211
C09896=1039.251,29.976,-85.294,169.373,38.362,157.210
C09897=1039.245,29.726,-85.278,169.371,38.362,157.210
C09898=1039.238,29.477,-85.263,169.369,38.361,157.210
C09899=1039.233,29.228,-85.246,169.367,38.361,157.210
C09900=1039.225,28.941,-85.227,169.365,38.360,157.210
C09901=1039.218,28.654,-85.209,169.362,38.360,157.210
C09902=1039.211,28.368,-85.190,169.360,38.358,157.209
C09903=1039.203,28.081,-85.172,169.357,38.358,157.209
C09904=1039.197,27.832,-85.155,169.355,38.358,157.209
C09905=1039.190,27.582,-85.139,169.353,38.358,157.209
C09906=1039.184,27.333,-85.123,169.352,38.357,157.209
C09907=1039.178,27.084,-85.107,169.350,38.356,157.209
C09908=1039.172,26.834,-85.092,169.348,38.356,157.209
C09909=1039.166,26.585,-85.076,169.345,38.355,157.209
C09910=1039.159,26.335,-85.059,169.343,38.355,157.208
C09911=1039.153,26.086,-85.043,169.341,38.355,157.208
C09912=1039.147,25.836,-85.027,169.339,38.354,157.208
C09913=1039.140,25.587,-85.011,169.337,38.354,157.208
C09914=1039.133,25.337,-84.995,169.335,38.353,157.208
C09915=1039.127,25.088,-84.979,169.333,38.353,157.208
C09916=1039.121,24.839,-84.963,169.331,38.352,157.208
C09917=1039.114,24.590,-84.947,169.329,38.352,157.208
C09918=1039.108,24.340,-84.931,169.327,38.352,157.208
C09919=1039.103,24.090,-84.915,169.324,38.351,157.207
C09920=1039.095,23.841,-84.899,169.322,38.351,157.207
C09921=1039.089,23.591,-84.883,169.320,38.350,157.207
C09922=1039.083,23.342,-84.867,169.318,38.349,157.207
C09923=1039.077,23.093,-84.851,169.316,38.349,157.207
C09924=1039.070,22.844,-84.835,169.314,38.349,157.207
C09925=1039.064,22.595,-84.819,169.312,38.348,157.207
C09926=1039.057,22.344,-84.804,169.310,38.348,157.206
C09927=1039.051,22.095,-84.788,169.308,38.347,157.206
C09928=1039.044,21.846,-84.772,169.307,38.347,157.206
C09929=1039.038,21.596,-84.756,169.304,38.346,157.206
C09930=1039.032,21.347,-84.740,169.302,38.346,157.206
C09931=1039.026,21.097,-84.724,169.300,38.345,157.206
C09932=1039.019,20.848,-84.709,169.298,38.345,157.206
C09933=1039.013,20.599,-84.693,169.296,38.345,157.206
C09934=1039.007,20.350,-84.677,169.294,38.344,157.205
C09935=1039.001,20.099,-84.661,169.292,38.344,157.205
C09936=1038.994,19.850,-84.645,169.290,38.343,157.205
C09937=1038.988,19.601,-84.629,169.288,38.342,157.205
C09938=1038.981,19.352,-84.613,169.286,38.343,157.205
C09939=1038.976,19.102,-84.598,169.283,38.342,157.205
C09940=1038.969,18.853,-84.582,169.281,38.342,157.205
C09941=1038.962,18.604,-84.567,169.279,38.341,157.205
C09942=1038.957,18.354,-84.551,169.277,38.340,157.204
C09943=1038.950,18.105,-84.535,169.275,38.341,157.204
C09944=1038.944,17.856,-84.519,169.273,38.340,157.204
C09945=1038.937,17.605,-84.504,169.271,38.339,157.204
C09946=1038.930,17.356,-84.488,169.269,38.339,157.204
C09947=1038.924,17.107,-84.472,169.267,38.338,157.204
C09948=1038.918,16.857,-84.457,169.265,38.338,157.204
C09949=1038.911,16.608,-84.441,169.262,38.338,157.204
C09950=1038.906,16.358,-84.426,169.260,38.337,157.203
C09951=1038.899,16.109,-84.410,169.258,38.337,157.203
C09952=1038.893,15.860,-84.394,169.256,38.336,157.203
C09953=1038.887,15.610,-84.379,169.254,38.336,157.203
C09954=1038.880,15.361,-84.363,169.252,38.336,157.203
C09955=1038.874,15.111,-84.348,169.250,38.335,157.203
C09956=1038.868,14.862,-84.332,169.248,38.335,157.203
C09957=1038.861,14.612,-84.317,169.246,38.334,157.203
C09958=1038.855,14.363,-84.301,169.244,38.334,157.202
C09959=1038.848,14.114,-84.285,169.242,38.334,157.202
C09960=1038.842,13.864,-84.270,169.239,38.333,157.202
C09961=1038.836,13.615,-84.255,169.237,38.333,157.202
C09962=1038.830,13.365,-84.239,169.235,38.332,157.202
C09963=1038.823,13.116,-84.224,169.233,38.332,157.202
C09964=1038.816,12.830,-84.206,169.231,38.332,157.202
C09965=1038.808,12.545,-84.189,169.228,38.331,157.202
C09966=1038.801,12.260,-84.171,169.226,38.331,157.202
C09967=1038.794,11.974,-84.154,169.224,38.331,157.202
C09968=1038.787,11.725,-84.138,169.222,38.330,157.201
C09969=1038.780,11.475,-84.123,169.220,38.330,157.201
C09970=1038.774,11.226,-84.108,169.218,38.330,157.201
C09971=1038.768,10.976,-84.092,169.215,38.329,157.201
C09972=1038.762,10.727,-84.077,169.213,38.329,157.201
C09973=1038.755,10.478,-84.062,169.210,38.329,157.201
C09974=1038.749,10.228,-84.047,169.208,38.328,157.201
C09975=1038.742,9.979,-84.031,169.206,38.328,157.201
C09976=1038.736,9.729,-84.016,169.204,38.328,157.201
C09977=1038.729,9.480,-84.001,169.202,38.327,157.200
C09978=1038.723,9.231,-83.985,169.200,38.327,157.200
C09979=1038.716,8.981,-83.971,169.198,38.327,157.200
C09980=1038.710,8.731,-83.956,169.196,38.326,157.200
C09981=1038.704,8.482,-83.939,169.194,38.326,157.200
C09982=1038.697,8.232,-83.924,169.191,38.325,157.200
C09983=1038.691,7.983,-83.909,169.189,38.325,157.200
C09984=1038.684,7.734,-83.894,169.187,38.325,157.200
C09985=1038.678,7.484,-83.879,169.185,38.324,157.200
C09986=1038.672,7.234,-83.864,169.183,38.324,157.199
C09987=1038.665,6.985,-83.849,169.181,38.324,157.199
C09988=1038.659,6.736,-83.833,169.179,38.323,157.199
C09989=1038.652,6.486,-83.818,169.177,38.323,157.199
C09990=1038.646,6.237,-83.804,169.175,38.323,157.199
C09991=1038.640,5.987,-83.789,169.173,38.322,157.199
C09992=1038.633,5.738,-83.773,169.171,38.321,157.199
C09993=1038.627,5.489,-83.758,169.169,38.322,157.199
C09994=1038.621,5.239,-83.743,169.166,38.321,157.199
C09995=1038.615,4.989,-83.728,169.163,38.320,157.198
C09996=1038.608,4.739,-83.713,169.161,38.321,157.198
//INST
///DATE 2021/06/17 10:57
///ATTR SC,RW,RJ
////FRAME ROBOT
///GROUP1 RB1
NOP
MOVL C00000 V=800.0 PL=0
MOVL C00001 V=800.0 PL=0
MOVL C00002 V=800.0 PL=0
MOVL C00003 V=800.0 PL=0
MOVL C00004 V=800.0 PL=0
MOVL C00005 V=800.0 PL=0
MOVL C00006 V=800.0 PL=0
MOVL C00007 V=800.0 PL=0
MOVL C00008 V=800.0 PL=0
MOVL C00009 V=800.0 PL=0
MOVL C00010 V=800.0 PL=0
MOVL C00011 V=800.0 PL=0
MOVL C00012 V=800.0 PL=0
MOVL C00013 V=800.0 PL=0
MOVL C00014 V=800.0 PL=0
MOVL C00015 V=800.0 PL=0
MOVL C00016 V=800.0 PL=0
MOVL C00017 V=800.0 PL=0
MOVL C00018 V=800.0 PL=0
MOVL C00019 V=800.0 PL=0
MOVL C00020 V=800.0 PL=0
MOVL C00021 V=800.0 PL=0
MOVL C00022 V=800.0 PL=0
MOVL C00023 V=800.0 PL=0
MOVL C00024 V=800.0 PL=0
MOVL C00025 V=800.0 PL=0
MOVL C00026 V=800.0 PL=0
MOVL C00027 V=800.0 PL=0
MOVL C00028 V=800.0 PL=0
MOVL C00029 V=800.0 PL=0
MOVL C00030 V=800.0 PL=0
MOVL C00031 V=800.0 PL=0
MOVL C00032 V=800.0 PL=0
MOVL C00033 V=800.0 PL=0
MOVL C00034 V=800.0 PL=0
MOVL C00035 V=800.0 PL=0
MOVL C00036 V=800.0 PL=0
MOVL C00037 V=800.0 PL=0
MOVL C00038 V=800.0 PL=0
MOVL C00039 V=800.0 PL=0
MOVL C00040 V=800.0 PL=0
MOVL C00041 V=800.0 PL=0
MOVL C00042 V=800.0 PL=0
MOVL C00043 V=800.0 PL=0
MOVL C00044 V=800.0 PL=0
MOVL C00045 V=800.0 PL=0
MOVL C00046 V=800.0 PL=0
MOVL C00047 V=800.0 PL=0
MOVL C00048 V=800.0 PL=0
MOVL C00049 V=800.0 PL=0
MOVL C00050 V=800.0 PL=0
MOVL C00051 V=800.0 PL=0
MOVL C00052 V=800.0 PL=0
MOVL C00053 V=800.0 PL=0
MOVL C00054 V=800.0 PL=0
MOVL C00055 V=800.0 PL=0
MOVL C00056 V=800.0 PL=0
MOVL C00057 V=800.0 PL=0
MOVL C00058 V=800.0 PL=0
MOVL C00059 V=800.0 PL=0
MOVL C00060 V=800.0 PL=0
MOVL C00061 V=800.0 PL=0
MOVL C00062 V=800.0 PL=0
MOVL C00063 V=800.0 PL=0
MOVL C00064 V=800.0 PL=0
MOVL C00065 V=800.0 PL=0
MOVL C00066 V=800.0 PL=0
MOVL C00067 V=800.0 PL=0
MOVL C00068 V=800.0 PL=0
MOVL C00069 V=800.0 PL=0
MOVL C00070 V=800.0 PL=0
MOVL C00071 V=800.0 PL=0
MOVL C00072 V=800.0 PL=0
MOVL C00073 V=800.0 PL=0
MOVL C00074 V=800.0 PL=0
MOVL C00075 V=800.0 PL=0
MOVL C00076 V=800.0 PL=0
MOVL C00077 V=800.0 PL=0
MOVL C00078 V=800.0 PL=0
MOVL C00079 V=800.0 PL=0
MOVL C00080 V=800.0 PL=0
MOVL C00081 V=800.0 PL=0
MOVL C00082 V=800.0 PL=0
MOVL C00083 V=800.0 PL=0
MOVL C00084 V=800.0 PL=0
MOVL C00085 V=800.0 PL=0
MOVL C00086 V=800.0 PL=0
MOVL C00087 V=800.0 PL=0
MOVL C00088 V=800.0 PL=0
MOVL C00089 V=800.0 PL=0
MOVL C00090 V=800.0 PL=0
MOVL C00091 V=800.0 PL=0
MOVL C00092 V=800.0 PL=0
MOVL C00093 V=800.0 PL=0
MOVL C00094 V=800.0 PL=0
MOVL C00095 V=800.0 PL=0
MOVL C00096 V=800.0 PL=0
MOVL C00097 V=800.0 PL=0
MOVL C00098 V=800.0 PL=0
MOVL C00099 V=800.0 PL=0
MOVL C00100 V=800.0 PL=0
MOVL C00101 V=800.0 PL=0
MOVL C00102 V=800.0 PL=0
MOVL C00103 V=800.0 PL=0
MOVL C00104 V=800.0 PL=0
MOVL C00105 V=800.0 PL=0
MOVL C00106 V=800.0 PL=0
MOVL C00107 V=800.0 PL=0
MOVL C00108 V=800.0 PL=0
MOVL C00109 V=800.0 PL=0
MOVL C00110 V=800.0 PL=0
MOVL C00111 V=800.0 PL=0
MOVL C00112 V=800.0 PL=0
MOVL C00113 V=800.0 PL=0
MOVL C00114 V=800.0 PL=0
MOVL C00115 V=800.0 PL=0
MOVL C00116 V=800.0 PL=0
MOVL C00117 V=800.0 PL=0
MOVL C00118 V=800.0 PL=0
MOVL C00119 V=800.0 PL=0
MOVL C00120 V=800.0 PL=0
MOVL C00121 V=800.0 PL=0
MOVL C00122 V=800.0 PL=0
MOVL C00123 V=800.0 PL=0
MOVL C00124 V=800.0 PL=0
MOVL C00125 V=800.0 PL=0
MOVL C00126 V=800.0 PL=0
MOVL C00127 V=800.0 PL=0
MOVL C00128 V=800.0 PL=0
MOVL C00129 V=800.0 PL=0
MOVL C00130 V=800.0 PL=0
MOVL C00131 V=800.0 PL=0
MOVL C00132 V=800.0 PL=0
MOVL C00133 V=800.0 PL=0
MOVL C00134 V=800.0 PL=0
MOVL C00135 V=800.0 PL=0
MOVL C00136 V=800.0 PL=0
MOVL C00137 V=800.0 PL=0
MOVL C00138 V=800.0 PL=0
MOVL C00139 V=800.0 PL=0
MOVL C00140 V=800.0 PL=0
MOVL C00141 V=800.0 PL=0
MOVL C00142 V=800.0 PL=0
MOVL C00143 V=800.0 PL=0
MOVL C00144 V=800.0 PL=0
MOVL C00145 V=800.0 PL=0
MOVL C00146 V=800.0 PL=0
MOVL C00147 V=800.0 PL=0
MOVL C00148 V=800.0 PL=0
MOVL C00149 V=800.0 PL=0
MOVL C00150 V=800.0 PL=0
MOVL C00151 V=800.0 PL=0
MOVL C00152 V=800.0 PL=0
MOVL C00153 V=800.0 PL=0
MOVL C00154 V=800.0 PL=0
MOVL C00155 V=800.0 PL=0
MOVL C00156 V=800.0 PL=0
MOVL C00157 V=800.0 PL=0
MOVL C00158 V=800.0 PL=0
MOVL C00159 V=800.0 PL=0
MOVL C00160 V=800.0 PL=0
MOVL C00161 V=800.0 PL=0
MOVL C00162 V=800.0 PL=0
MOVL C00163 V=800.0 PL=0
MOVL C00164 V=800.0 PL=0
MOVL C00165 V=800.0 PL=0
MOVL C00166 V=800.0 PL=0
MOVL C00167 V=800.0 PL=0
MOVL C00168 V=800.0 PL=0
MOVL C00169 V=800.0 PL=0
MOVL C00170 V=800.0 PL=0
MOVL C00171 V=800.0 PL=0
MOVL C00172 V=800.0 PL=0
MOVL C00173 V=800.0 PL=0
MOVL C00174 V=800.0 PL=0
MOVL C00175 V=800.0 PL=0
MOVL C00176 V=800.0 PL=0
MOVL C00177 V=800.0 PL=0
MOVL C00178 V=800.0 PL=0
MOVL C00179 V=800.0 PL=0
MOVL C00180 V=800.0 PL=0
MOVL C00181 V=800.0 PL=0
MOVL C00182 V=800.0 PL=0
MOVL C00183 V=800.0 PL=0
MOVL C00184 V=800.0 PL=0
MOVL C00185 V=800.0 PL=0
MOVL C00186 V=800.0 PL=0
MOVL C00187 V=800.0 PL=0
MOVL C00188 V=800.0 PL=0
MOVL C00189 V=800.0 PL=0
MOVL C00190 V=800.0 PL=0
MOVL C00191 V=800.0 PL=0
MOVL C00192 V=800.0 PL=0
MOVL C00193 V=800.0 PL=0
MOVL C00194 V=800.0 PL=0
MOVL C00195 V=800.0 PL=0
MOVL C00196 V=800.0 PL=0
MOVL C00197 V=800.0 PL=0
MOVL C00198 V=800.0 PL=0
MOVL C00199 V=800.0 PL=0
MOVL C00200 V=800.0 PL=0
MOVL C00201 V=800.0 PL=0
MOVL C00202 V=800.0 PL=0
MOVL C00203 V=800.0 PL=0
MOVL C00204 V=800.0 PL=0
MOVL C00205 V=800.0 PL=0
MOVL C00206 V=800.0 PL=0
MOVL C00207 V=800.0 PL=0
MOVL C00208 V=800.0 PL=0
MOVL C00209 V=800.0 PL=0
MOVL C00210 V=800.0 PL=0
MOVL C00211 V=800.0 PL=0
MOVL C00212 V=800.0 PL=0
MOVL C00213 V=800.0 PL=0
MOVL C00214 V=800.0 PL=0
MOVL C00215 V=800.0 PL=0
MOVL C00216 V=800.0 PL=0
MOVL C00217 V=800.0 PL=0
MOVL C00218 V=800.0 PL=0
MOVL C00219 V=800.0 PL=0
MOVL C00220 V=800.0 PL=0
MOVL C00221 V=800.0 PL=0
MOVL C00222 V=800.0 PL=0
MOVL C00223 V=800.0 PL=0
MOVL C00224 V=800.0 PL=0
MOVL C00225 V=800.0 PL=0
MOVL C00226 V=800.0 PL=0
MOVL C00227 V=800.0 PL=0
MOVL C00228 V=800.0 PL=0
MOVL C00229 V=800.0 PL=0
MOVL C00230 V=800.0 PL=0
MOVL C00231 V=800.0 PL=0
MOVL C00232 V=800.0 PL=0
MOVL C00233 V=800.0 PL=0
MOVL C00234 V=800.0 PL=0
MOVL C00235 V=800.0 PL=0
MOVL C00236 V=800.0 PL=0
MOVL C00237 V=800.0 PL=0
MOVL C00238 V=800.0 PL=0
MOVL C00239 V=800.0 PL=0
MOVL C00240 V=800.0 PL=0
MOVL C00241 V=800.0 PL=0
MOVL C00242 V=800.0 PL=0
MOVL C00243 V=800.0 PL=0
MOVL C00244 V=800.0 PL=0
MOVL C00245 V=800.0 PL=0
MOVL C00246 V=800.0 PL=0
MOVL C00247 V=800.0 PL=0
MOVL C00248 V=800.0 PL=0
MOVL C00249 V=800.0 PL=0
MOVL C00250 V=800.0 PL=0
MOVL C00251 V=800.0 PL=0
MOVL C00252 V=800.0 PL=0
MOVL C00253 V=800.0 PL=0
MOVL C00254 V=800.0 PL=0
MOVL C00255 V=800.0 PL=0
MOVL C00256 V=800.0 PL=0
MOVL C00257 V=800.0 PL=0
MOVL C00258 V=800.0 PL=0
MOVL C00259 V=800.0 PL=0
MOVL C00260 V=800.0 PL=0
MOVL C00261 V=800.0 PL=0
MOVL C00262 V=800.0 PL=0
MOVL C00263 V=800.0 PL=0
MOVL C00264 V=800.0 PL=0
MOVL C00265 V=800.0 PL=0
MOVL C00266 V=800.0 PL=0
MOVL C00267 V=800.0 PL=0
MOVL C00268 V=800.0 PL=0
MOVL C00269 V=800.0 PL=0
MOVL C00270 V=800.0 PL=0
MOVL C00271 V=800.0 PL=0
MOVL C00272 V=800.0 PL=0
MOVL C00273 V=800.0 PL=0
MOVL C00274 V=800.0 PL=0
MOVL C00275 V=800.0 PL=0
MOVL C00276 V=800.0 PL=0
MOVL C00277 V=800.0 PL=0
MOVL C00278 V=800.0 PL=0
MOVL C00279 V=800.0 PL=0
MOVL C00280 V=800.0 PL=0
MOVL C00281 V=800.0 PL=0
MOVL C00282 V=800.0 PL=0
MOVL C00283 V=800.0 PL=0
MOVL C00284 V=800.0 PL=0
MOVL C00285 V=800.0 PL=0
MOVL C00286 V=800.0 PL=0
MOVL C00287 V=800.0 PL=0
MOVL C00288 V=800.0 PL=0
MOVL C00289 V=800.0 PL=0
MOVL C00290 V=800.0 PL=0
MOVL C00291 V=800.0 PL=0
MOVL C00292 V=800.0 PL=0
MOVL C00293 V=800.0 PL=0
MOVL C00294 V=800.0 PL=0
MOVL C00295 V=800.0 PL=0
MOVL C00296 V=800.0 PL=0
MOVL C00297 V=800.0 PL=0
MOVL C00298 V=800.0 PL=0
MOVL C00299 V=800.0 PL=0
MOVL C00300 V=800.0 PL=0
MOVL C00301 V=800.0 PL=0
MOVL C00302 V=800.0 PL=0
MOVL C00303 V=800.0 PL=0
MOVL C00304 V=800.0 PL=0
MOVL C00305 V=800.0 PL=0
MOVL C00306 V=800.0 PL=0
MOVL C00307 V=800.0 PL=0
MOVL C00308 V=800.0 PL=0
MOVL C00309 V=800.0 PL=0
MOVL C00310 V=800.0 PL=0
MOVL C00311 V=800.0 PL=0
MOVL C00312 V=800.0 PL=0
MOVL C00313 V=800.0 PL=0
MOVL C00314 V=800.0 PL=0
MOVL C00315 V=800.0 PL=0
MOVL C00316 V=800.0 PL=0
MOVL C00317 V=800.0 PL=0
MOVL C00318 V=800.0 PL=0
MOVL C00319 V=800.0 PL=0
MOVL C00320 V=800.0 PL=0
MOVL C00321 V=800.0 PL=0
MOVL C00322 V=800.0 PL=0
MOVL C00323 V=800.0 PL=0
MOVL C00324 V=800.0 PL=0
MOVL C00325 V=800.0 PL=0
MOVL C00326 V=800.0 PL=0
MOVL C00327 V=800.0 PL=0
MOVL C00328 V=800.0 PL=0
MOVL C00329 V=800.0 PL=0
MOVL C00330 V=800.0 PL=0
MOVL C00331 V=800.0 PL=0
MOVL C00332 V=800.0 PL=0
MOVL C00333 V=800.0 PL=0
MOVL C00334 V=800.0 PL=0
MOVL C00335 V=800.0 PL=0
MOVL C00336 V=800.0 PL=0
MOVL C00337 V=800.0 PL=0
MOVL C00338 V=800.0 PL=0
MOVL C00339 V=800.0 PL=0
MOVL C00340 V=800.0 PL=0
MOVL C00341 V=800.0 PL=0
MOVL C00342 V=800.0 PL=0
MOVL C00343 V=800.0 PL=0
MOVL C00344 V=800.0 PL=0
MOVL C00345 V=800.0 PL=0
MOVL C00346 V=800.0 PL=0
MOVL C00347 V=800.0 PL=0
MOVL C00348 V=800.0 PL=0
MOVL C00349 V=800.0 PL=0
MOVL C00350 V=800.0 PL=0
MOVL C00351 V=800.0 PL=0
MOVL C00352 V=800.0 PL=0
MOVL C00353 V=800.0 PL=0
MOVL C00354 V=800.0 PL=0
MOVL C00355 V=800.0 PL=0
MOVL C00356 V=800.0 PL=0
MOVL C00357 V=800.0 PL=0
MOVL C00358 V=800.0 PL=0
MOVL C00359 V=800.0 PL=0
MOVL C00360 V=800.0 PL=0
MOVL C00361 V=800.0 PL=0
MOVL C00362 V=800.0 PL=0
MOVL C00363 V=800.0 PL=0
MOVL C00364 V=800.0 PL=0
MOVL C00365 V=800.0 PL=0
MOVL C00366 V=800.0 PL=0
MOVL C00367 V=800.0 PL=0
MOVL C00368 V=800.0 PL=0
MOVL C00369 V=800.0 PL=0
MOVL C00370 V=800.0 PL=0
MOVL C00371 V=800.0 PL=0
MOVL C00372 V=800.0 PL=0
MOVL C00373 V=800.0 PL=0
MOVL C00374 V=800.0 PL=0
MOVL C00375 V=800.0 PL=0
MOVL C00376 V=800.0 PL=0
MOVL C00377 V=800.0 PL=0
MOVL C00378 V=800.0 PL=0
MOVL C00379 V=800.0 PL=0
MOVL C00380 V=800.0 PL=0
MOVL C00381 V=800.0 PL=0
MOVL C00382 V=800.0 PL=0
MOVL C00383 V=800.0 PL=0
MOVL C00384 V=800.0 PL=0
MOVL C00385 V=800.0 PL=0
MOVL C00386 V=800.0 PL=0
MOVL C00387 V=800.0 PL=0
MOVL C00388 V=800.0 PL=0
MOVL C00389 V=800.0 PL=0
MOVL C00390 V=800.0 PL=0
MOVL C00391 V=800.0 PL=0
MOVL C00392 V=800.0 PL=0
MOVL C00393 V=800.0 PL=0
MOVL C00394 V=800.0 PL=0
MOVL C00395 V=800.0 PL=0
MOVL C00396 V=800.0 PL=0
MOVL C00397 V=800.0 PL=0
MOVL C00398 V=800.0 PL=0
MOVL C00399 V=800.0 PL=0
MOVL C00400 V=800.0 PL=0
MOVL C00401 V=800.0 PL=0
MOVL C00402 V=800.0 PL=0
MOVL C00403 V=800.0 PL=0
MOVL C00404 V=800.0 PL=0
MOVL C00405 V=800.0 PL=0
MOVL C00406 V=800.0 PL=0
MOVL C00407 V=800.0 PL=0
MOVL C00408 V=800.0 PL=0
MOVL C00409 V=800.0 PL=0
MOVL C00410 V=800.0 PL=0
MOVL C00411 V=800.0 PL=0
MOVL C00412 V=800.0 PL=0
MOVL C00413 V=800.0 PL=0
MOVL C00414 V=800.0 PL=0
MOVL C00415 V=800.0 PL=0
MOVL C00416 V=800.0 PL=0
MOVL C00417 V=800.0 PL=0
MOVL C00418 V=800.0 PL=0
MOVL C00419 V=800.0 PL=0
MOVL C00420 V=800.0 PL=0
MOVL C00421 V=800.0 PL=0
MOVL C00422 V=800.0 PL=0
MOVL C00423 V=800.0 PL=0
MOVL C00424 V=800.0 PL=0
MOVL C00425 V=800.0 PL=0
MOVL C00426 V=800.0 PL=0
MOVL C00427 V=800.0 PL=0
MOVL C00428 V=800.0 PL=0
MOVL C00429 V=800.0 PL=0
MOVL C00430 V=800.0 PL=0
MOVL C00431 V=800.0 PL=0
MOVL C00432 V=800.0 PL=0
MOVL C00433 V=800.0 PL=0
MOVL C00434 V=800.0 PL=0
MOVL C00435 V=800.0 PL=0
MOVL C00436 V=800.0 PL=0
MOVL C00437 V=800.0 PL=0
MOVL C00438 V=800.0 PL=0
MOVL C00439 V=800.0 PL=0
MOVL C00440 V=800.0 PL=0
MOVL C00441 V=800.0 PL=0
MOVL C00442 V=800.0 PL=0
MOVL C00443 V=800.0 PL=0
MOVL C00444 V=800.0 PL=0
MOVL C00445 V=800.0 PL=0
MOVL C00446 V=800.0 PL=0
MOVL C00447 V=800.0 PL=0
MOVL C00448 V=800.0 PL=0
MOVL C00449 V=800.0 PL=0
MOVL C00450 V=800.0 PL=0
MOVL C00451 V=800.0 PL=0
MOVL C00452 V=800.0 PL=0
MOVL C00453 V=800.0 PL=0
MOVL C00454 V=800.0 PL=0
MOVL C00455 V=800.0 PL=0
MOVL C00456 V=800.0 PL=0
MOVL C00457 V=800.0 PL=0
MOVL C00458 V=800.0 PL=0
MOVL C00459 V=800.0 PL=0
MOVL C00460 V=800.0 PL=0
MOVL C00461 V=800.0 PL=0
MOVL C00462 V=800.0 PL=0
MOVL C00463 V=800.0 PL=0
MOVL C00464 V=800.0 PL=0
MOVL C00465 V=800.0 PL=0
MOVL C00466 V=800.0 PL=0
MOVL C00467 V=800.0 PL=0
MOVL C00468 V=800.0 PL=0
MOVL C00469 V=800.0 PL=0
MOVL C00470 V=800.0 PL=0
MOVL C00471 V=800.0 PL=0
MOVL C00472 V=800.0 PL=0
MOVL C00473 V=800.0 PL=0
MOVL C00474 V=800.0 PL=0
MOVL C00475 V=800.0 PL=0
MOVL C00476 V=800.0 PL=0
MOVL C00477 V=800.0 PL=0
MOVL C00478 V=800.0 PL=0
MOVL C00479 V=800.0 PL=0
MOVL C00480 V=800.0 PL=0
MOVL C00481 V=800.0 PL=0
MOVL C00482 V=800.0 PL=0
MOVL C00483 V=800.0 PL=0
MOVL C00484 V=800.0 PL=0
MOVL C00485 V=800.0 PL=0
MOVL C00486 V=800.0 PL=0
MOVL C00487 V=800.0 PL=0
MOVL C00488 V=800.0 PL=0
MOVL C00489 V=800.0 PL=0
MOVL C00490 V=800.0 PL=0
MOVL C00491 V=800.0 PL=0
MOVL C00492 V=800.0 PL=0
MOVL C00493 V=800.0 PL=0
MOVL C00494 V=800.0 PL=0
MOVL C00495 V=800.0 PL=0
MOVL C00496 V=800.0 PL=0
MOVL C00497 V=800.0 PL=0
MOVL C00498 V=800.0 PL=0
MOVL C00499 V=800.0 PL=0
MOVL C00500 V=800.0 PL=0
MOVL C00501 V=800.0 PL=0
MOVL C00502 V=800.0 PL=0
MOVL C00503 V=800.0 PL=0
MOVL C00504 V=800.0 PL=0
MOVL C00505 V=800.0 PL=0
MOVL C00506 V=800.0 PL=0
MOVL C00507 V=800.0 PL=0
MOVL C00508 V=800.0 PL=0
MOVL C00509 V=800.0 PL=0
MOVL C00510 V=800.0 PL=0
MOVL C00511 V=800.0 PL=0
MOVL C00512 V=800.0 PL=0
MOVL C00513 V=800.0 PL=0
MOVL C00514 V=800.0 PL=0
MOVL C00515 V=800.0 PL=0
MOVL C00516 V=800.0 PL=0
MOVL C00517 V=800.0 PL=0
MOVL C00518 V=800.0 PL=0
MOVL C00519 V=800.0 PL=0
MOVL C00520 V=800.0 PL=0
MOVL C00521 V=800.0 PL=0
MOVL C00522 V=800.0 PL=0
MOVL C00523 V=800.0 PL=0
MOVL C00524 V=800.0 PL=0
MOVL C00525 V=800.0 PL=0
MOVL C00526 V=800.0 PL=0
MOVL C00527 V=800.0 PL=0
MOVL C00528 V=800.0 PL=0
MOVL C00529 V=800.0 PL=0
MOVL C00530 V=800.0 PL=0
MOVL C00531 V=800.0 PL=0
MOVL C00532 V=800.0 PL=0
MOVL C00533 V=800.0 PL=0
MOVL C00534 V=800.0 PL=0
MOVL C00535 V=800.0 PL=0
MOVL C00536 V=800.0 PL=0
MOVL C00537 V=800.0 PL=0
MOVL C00538 V=800.0 PL=0
MOVL C00539 V=800.0 PL=0
MOVL C00540 V=800.0 PL=0
MOVL C00541 V=800.0 PL=0
MOVL C00542 V=800.0 PL=0
MOVL C00543 V=800.0 PL=0
MOVL C00544 V=800.0 PL=0
MOVL C00545 V=800.0 PL=0
MOVL C00546 V=800.0 PL=0
MOVL C00547 V=800.0 PL=0
MOVL C00548 V=800.0 PL=0
MOVL C00549 V=800.0 PL=0
MOVL C00550 V=800.0 PL=0
MOVL C00551 V=800.0 PL=0
MOVL C00552 V=800.0 PL=0
MOVL C00553 V=800.0 PL=0
MOVL C00554 V=800.0 PL=0
MOVL C00555 V=800.0 PL=0
MOVL C00556 V=800.0 PL=0
MOVL C00557 V=800.0 PL=0
MOVL C00558 V=800.0 PL=0
MOVL C00559 V=800.0 PL=0
MOVL C00560 V=800.0 PL=0
MOVL C00561 V=800.0 PL=0
MOVL C00562 V=800.0 PL=0
MOVL C00563 V=800.0 PL=0
MOVL C00564 V=800.0 PL=0
MOVL C00565 V=800.0 PL=0
MOVL C00566 V=800.0 PL=0
MOVL C00567 V=800.0 PL=0
MOVL C00568 V=800.0 PL=0
MOVL C00569 V=800.0 PL=0
MOVL C00570 V=800.0 PL=0
MOVL C00571 V=800.0 PL=0
MOVL C00572 V=800.0 PL=0
MOVL C00573 V=800.0 PL=0
MOVL C00574 V=800.0 PL=0
MOVL C00575 V=800.0 PL=0
MOVL C00576 V=800.0 PL=0
MOVL C00577 V=800.0 PL=0
MOVL C00578 V=800.0 PL=0
MOVL C00579 V=800.0 PL=0
MOVL C00580 V=800.0 PL=0
MOVL C00581 V=800.0 PL=0
MOVL C00582 V=800.0 PL=0
MOVL C00583 V=800.0 PL=0
MOVL C00584 V=800.0 PL=0
MOVL C00585 V=800.0 PL=0
MOVL C00586 V=800.0 PL=0
MOVL C00587 V=800.0 PL=0
MOVL C00588 V=800.0 PL=0
MOVL C00589 V=800.0 PL=0
MOVL C00590 V=800.0 PL=0
MOVL C00591 V=800.0 PL=0
MOVL C00592 V=800.0 PL=0
MOVL C00593 V=800.0 PL=0
MOVL C00594 V=800.0 PL=0
MOVL C00595 V=800.0 PL=0
MOVL C00596 V=800.0 PL=0
MOVL C00597 V=800.0 PL=0
MOVL C00598 V=800.0 PL=0
MOVL C00599 V=800.0 PL=0
MOVL C00600 V=800.0 PL=0
MOVL C00601 V=800.0 PL=0
MOVL C00602 V=800.0 PL=0
MOVL C00603 V=800.0 PL=0
MOVL C00604 V=800.0 PL=0
MOVL C00605 V=800.0 PL=0
MOVL C00606 V=800.0 PL=0
MOVL C00607 V=800.0 PL=0
MOVL C00608 V=800.0 PL=0
MOVL C00609 V=800.0 PL=0
MOVL C00610 V=800.0 PL=0
MOVL C00611 V=800.0 PL=0
MOVL C00612 V=800.0 PL=0
MOVL C00613 V=800.0 PL=0
MOVL C00614 V=800.0 PL=0
MOVL C00615 V=800.0 PL=0
MOVL C00616 V=800.0 PL=0
MOVL C00617 V=800.0 PL=0
MOVL C00618 V=800.0 PL=0
MOVL C00619 V=800.0 PL=0
MOVL C00620 V=800.0 PL=0
MOVL C00621 V=800.0 PL=0
MOVL C00622 V=800.0 PL=0
MOVL C00623 V=800.0 PL=0
MOVL C00624 V=800.0 PL=0
MOVL C00625 V=800.0 PL=0
MOVL C00626 V=800.0 PL=0
MOVL C00627 V=800.0 PL=0
MOVL C00628 V=800.0 PL=0
MOVL C00629 V=800.0 PL=0
MOVL C00630 V=800.0 PL=0
MOVL C00631 V=800.0 PL=0
MOVL C00632 V=800.0 PL=0
MOVL C00633 V=800.0 PL=0
MOVL C00634 V=800.0 PL=0
MOVL C00635 V=800.0 PL=0
MOVL C00636 V=800.0 PL=0
MOVL C00637 V=800.0 PL=0
MOVL C00638 V=800.0 PL=0
MOVL C00639 V=800.0 PL=0
MOVL C00640 V=800.0 PL=0
MOVL C00641 V=800.0 PL=0
MOVL C00642 V=800.0 PL=0
MOVL C00643 V=800.0 PL=0
MOVL C00644 V=800.0 PL=0
MOVL C00645 V=800.0 PL=0
MOVL C00646 V=800.0 PL=0
MOVL C00647 V=800.0 PL=0
MOVL C00648 V=800.0 PL=0
MOVL C00649 V=800.0 PL=0
MOVL C00650 V=800.0 PL=0
MOVL C00651 V=800.0 PL=0
MOVL C00652 V=800.0 PL=0
MOVL C00653 V=800.0 PL=0
MOVL C00654 V=800.0 PL=0
MOVL C00655 V=800.0 PL=0
MOVL C00656 V=800.0 PL=0
MOVL C00657 V=800.0 PL=0
MOVL C00658 V=800.0 PL=0
MOVL C00659 V=800.0 PL=0
MOVL C00660 V=800.0 PL=0
MOVL C00661 V=800.0 PL=0
MOVL C00662 V=800.0 PL=0
MOVL C00663 V=800.0 PL=0
MOVL C00664 V=800.0 PL=0
MOVL C00665 V=800.0 PL=0
MOVL C00666 V=800.0 PL=0
MOVL C00667 V=800.0 PL=0
MOVL C00668 V=800.0 PL=0
MOVL C00669 V=800.0 PL=0
MOVL C00670 V=800.0 PL=0
MOVL C00671 V=800.0 PL=0
MOVL C00672 V=800.0 PL=0
MOVL C00673 V=800.0 PL=0
MOVL C00674 V=800.0 PL=0
MOVL C00675 V=800.0 PL=0
MOVL C00676 V=800.0 PL=0
MOVL C00677 V=800.0 PL=0
MOVL C00678 V=800.0 PL=0
MOVL C00679 V=800.0 PL=0
MOVL C00680 V=800.0 PL=0
MOVL C00681 V=800.0 PL=0
MOVL C00682 V=800.0 PL=0
MOVL C00683 V=800.0 PL=0
MOVL C00684 V=800.0 PL=0
MOVL C00685 V=800.0 PL=0
MOVL C00686 V=800.0 PL=0
MOVL C00687 V=800.0 PL=0
MOVL C00688 V=800.0 PL=0
MOVL C00689 V=800.0 PL=0
MOVL C00690 V=800.0 PL=0
MOVL C00691 V=800.0 PL=0
MOVL C00692 V=800.0 PL=0
MOVL C00693 V=800.0 PL=0
MOVL C00694 V=800.0 PL=0
MOVL C00695 V=800.0 PL=0
MOVL C00696 V=800.0 PL=0
MOVL C00697 V=800.0 PL=0
MOVL C00698 V=800.0 PL=0
MOVL C00699 V=800.0 PL=0
MOVL C00700 V=800.0 PL=0
MOVL C00701 V=800.0 PL=0
MOVL C00702 V=800.0 PL=0
MOVL C00703 V=800.0 PL=0
MOVL C00704 V=800.0 PL=0
MOVL C00705 V=800.0 PL=0
MOVL C00706 V=800.0 PL=0
MOVL C00707 V=800.0 PL=0
MOVL C00708 V=800.0 PL=0
MOVL C00709 V=800.0 PL=0
MOVL C00710 V=800.0 PL=0
MOVL C00711 V=800.0 PL=0
MOVL C00712 V=800.0 PL=0
MOVL C00713 V=800.0 PL=0
MOVL C00714 V=800.0 PL=0
MOVL C00715 V=800.0 PL=0
MOVL C00716 V=800.0 PL=0
MOVL C00717 V=800.0 PL=0
MOVL C00718 V=800.0 PL=0
MOVL C00719 V=800.0 PL=0
MOVL C00720 V=800.0 PL=0
MOVL C00721 V=800.0 PL=0
MOVL C00722 V=800.0 PL=0
MOVL C00723 V=800.0 PL=0
MOVL C00724 V=800.0 PL=0
MOVL C00725 V=800.0 PL=0
MOVL C00726 V=800.0 PL=0
MOVL C00727 V=800.0 PL=0
MOVL C00728 V=800.0 PL=0
MOVL C00729 V=800.0 PL=0
MOVL C00730 V=800.0 PL=0
MOVL C00731 V=800.0 PL=0
MOVL C00732 V=800.0 PL=0
MOVL C00733 V=800.0 PL=0
MOVL C00734 V=800.0 PL=0
MOVL C00735 V=800.0 PL=0
MOVL C00736 V=800.0 PL=0
MOVL C00737 V=800.0 PL=0
MOVL C00738 V=800.0 PL=0
MOVL C00739 V=800.0 PL=0
MOVL C00740 V=800.0 PL=0
MOVL C00741 V=800.0 PL=0
MOVL C00742 V=800.0 PL=0
MOVL C00743 V=800.0 PL=0
MOVL C00744 V=800.0 PL=0
MOVL C00745 V=800.0 PL=0
MOVL C00746 V=800.0 PL=0
MOVL C00747 V=800.0 PL=0
MOVL C00748 V=800.0 PL=0
MOVL C00749 V=800.0 PL=0
MOVL C00750 V=800.0 PL=0
MOVL C00751 V=800.0 PL=0
MOVL C00752 V=800.0 PL=0
MOVL C00753 V=800.0 PL=0
MOVL C00754 V=800.0 PL=0
MOVL C00755 V=800.0 PL=0
MOVL C00756 V=800.0 PL=0
MOVL C00757 V=800.0 PL=0
MOVL C00758 V=800.0 PL=0
MOVL C00759 V=800.0 PL=0
MOVL C00760 V=800.0 PL=0
MOVL C00761 V=800.0 PL=0
MOVL C00762 V=800.0 PL=0
MOVL C00763 V=800.0 PL=0
MOVL C00764 V=800.0 PL=0
MOVL C00765 V=800.0 PL=0
MOVL C00766 V=800.0 PL=0
MOVL C00767 V=800.0 PL=0
MOVL C00768 V=800.0 PL=0
MOVL C00769 V=800.0 PL=0
MOVL C00770 V=800.0 PL=0
MOVL C00771 V=800.0 PL=0
MOVL C00772 V=800.0 PL=0
MOVL C00773 V=800.0 PL=0
MOVL C00774 V=800.0 PL=0
MOVL C00775 V=800.0 PL=0
MOVL C00776 V=800.0 PL=0
MOVL C00777 V=800.0 PL=0
MOVL C00778 V=800.0 PL=0
MOVL C00779 V=800.0 PL=0
MOVL C00780 V=800.0 PL=0
MOVL C00781 V=800.0 PL=0
MOVL C00782 V=800.0 PL=0
MOVL C00783 V=800.0 PL=0
MOVL C00784 V=800.0 PL=0
MOVL C00785 V=800.0 PL=0
MOVL C00786 V=800.0 PL=0
MOVL C00787 V=800.0 PL=0
MOVL C00788 V=800.0 PL=0
MOVL C00789 V=800.0 PL=0
MOVL C00790 V=800.0 PL=0
MOVL C00791 V=800.0 PL=0
MOVL C00792 V=800.0 PL=0
MOVL C00793 V=800.0 PL=0
MOVL C00794 V=800.0 PL=0
MOVL C00795 V=800.0 PL=0
MOVL C00796 V=800.0 PL=0
MOVL C00797 V=800.0 PL=0
MOVL C00798 V=800.0 PL=0
MOVL C00799 V=800.0 PL=0
MOVL C00800 V=800.0 PL=0
MOVL C00801 V=800.0 PL=0
MOVL C00802 V=800.0 PL=0
MOVL C00803 V=800.0 PL=0
MOVL C00804 V=800.0 PL=0
MOVL C00805 V=800.0 PL=0
MOVL C00806 V=800.0 PL=0
MOVL C00807 V=800.0 PL=0
MOVL C00808 V=800.0 PL=0
MOVL C00809 V=800.0 PL=0
MOVL C00810 V=800.0 PL=0
MOVL C00811 V=800.0 PL=0
MOVL C00812 V=800.0 PL=0
MOVL C00813 V=800.0 PL=0
MOVL C00814 V=800.0 PL=0
MOVL C00815 V=800.0 PL=0
MOVL C00816 V=800.0 PL=0
MOVL C00817 V=800.0 PL=0
MOVL C00818 V=800.0 PL=0
MOVL C00819 V=800.0 PL=0
MOVL C00820 V=800.0 PL=0
MOVL C00821 V=800.0 PL=0
MOVL C00822 V=800.0 PL=0
MOVL C00823 V=800.0 PL=0
MOVL C00824 V=800.0 PL=0
MOVL C00825 V=800.0 PL=0
MOVL C00826 V=800.0 PL=0
MOVL C00827 V=800.0 PL=0
MOVL C00828 V=800.0 PL=0
MOVL C00829 V=800.0 PL=0
MOVL C00830 V=800.0 PL=0
MOVL C00831 V=800.0 PL=0
MOVL C00832 V=800.0 PL=0
MOVL C00833 V=800.0 PL=0
MOVL C00834 V=800.0 PL=0
MOVL C00835 V=800.0 PL=0
MOVL C00836 V=800.0 PL=0
MOVL C00837 V=800.0 PL=0
MOVL C00838 V=800.0 PL=0
MOVL C00839 V=800.0 PL=0
MOVL C00840 V=800.0 PL=0
MOVL C00841 V=800.0 PL=0
MOVL C00842 V=800.0 PL=0
MOVL C00843 V=800.0 PL=0
MOVL C00844 V=800.0 PL=0
MOVL C00845 V=800.0 PL=0
MOVL C00846 V=800.0 PL=0
MOVL C00847 V=800.0 PL=0
MOVL C00848 V=800.0 PL=0
MOVL C00849 V=800.0 PL=0
MOVL C00850 V=800.0 PL=0
MOVL C00851 V=800.0 PL=0
MOVL C00852 V=800.0 PL=0
MOVL C00853 V=800.0 PL=0
MOVL C00854 V=800.0 PL=0
MOVL C00855 V=800.0 PL=0
MOVL C00856 V=800.0 PL=0
MOVL C00857 V=800.0 PL=0
MOVL C00858 V=800.0 PL=0
MOVL C00859 V=800.0 PL=0
MOVL C00860 V=800.0 PL=0
MOVL C00861 V=800.0 PL=0
MOVL C00862 V=800.0 PL=0
MOVL C00863 V=800.0 PL=0
MOVL C00864 V=800.0 PL=0
MOVL C00865 V=800.0 PL=0
MOVL C00866 V=800.0 PL=0
MOVL C00867 V=800.0 PL=0
MOVL C00868 V=800.0 PL=0
MOVL C00869 V=800.0 PL=0
MOVL C00870 V=800.0 PL=0
MOVL C00871 V=800.0 PL=0
MOVL C00872 V=800.0 PL=0
MOVL C00873 V=800.0 PL=0
MOVL C00874 V=800.0 PL=0
MOVL C00875 V=800.0 PL=0
MOVL C00876 V=800.0 PL=0
MOVL C00877 V=800.0 PL=0
MOVL C00878 V=800.0 PL=0
MOVL C00879 V=800.0 PL=0
MOVL C00880 V=800.0 PL=0
MOVL C00881 V=800.0 PL=0
MOVL C00882 V=800.0 PL=0
MOVL C00883 V=800.0 PL=0
MOVL C00884 V=800.0 PL=0
MOVL C00885 V=800.0 PL=0
MOVL C00886 V=800.0 PL=0
MOVL C00887 V=800.0 PL=0
MOVL C00888 V=800.0 PL=0
MOVL C00889 V=800.0 PL=0
MOVL C00890 V=800.0 PL=0
MOVL C00891 V=800.0 PL=0
MOVL C00892 V=800.0 PL=0
MOVL C00893 V=800.0 PL=0
MOVL C00894 V=800.0 PL=0
MOVL C00895 V=800.0 PL=0
MOVL C00896 V=800.0 PL=0
MOVL C00897 V=800.0 PL=0
MOVL C00898 V=800.0 PL=0
MOVL C00899 V=800.0 PL=0
MOVL C00900 V=800.0 PL=0
MOVL C00901 V=800.0 PL=0
MOVL C00902 V=800.0 PL=0
MOVL C00903 V=800.0 PL=0
MOVL C00904 V=800.0 PL=0
MOVL C00905 V=800.0 PL=0
MOVL C00906 V=800.0 PL=0
MOVL C00907 V=800.0 PL=0
MOVL C00908 V=800.0 PL=0
MOVL C00909 V=800.0 PL=0
MOVL C00910 V=800.0 PL=0
MOVL C00911 V=800.0 PL=0
MOVL C00912 V=800.0 PL=0
MOVL C00913 V=800.0 PL=0
MOVL C00914 V=800.0 PL=0
MOVL C00915 V=800.0 PL=0
MOVL C00916 V=800.0 PL=0
MOVL C00917 V=800.0 PL=0
MOVL C00918 V=800.0 PL=0
MOVL C00919 V=800.0 PL=0
MOVL C00920 V=800.0 PL=0
MOVL C00921 V=800.0 PL=0
MOVL C00922 V=800.0 PL=0
MOVL C00923 V=800.0 PL=0
MOVL C00924 V=800.0 PL=0
MOVL C00925 V=800.0 PL=0
MOVL C00926 V=800.0 PL=0
MOVL C00927 V=800.0 PL=0
MOVL C00928 V=800.0 PL=0
MOVL C00929 V=800.0 PL=0
MOVL C00930 V=800.0 PL=0
MOVL C00931 V=800.0 PL=0
MOVL C00932 V=800.0 PL=0
MOVL C00933 V=800.0 PL=0
MOVL C00934 V=800.0 PL=0
MOVL C00935 V=800.0 PL=0
MOVL C00936 V=800.0 PL=0
MOVL C00937 V=800.0 PL=0
MOVL C00938 V=800.0 PL=0
MOVL C00939 V=800.0 PL=0
MOVL C00940 V=800.0 PL=0
MOVL C00941 V=800.0 PL=0
MOVL C00942 V=800.0 PL=0
MOVL C00943 V=800.0 PL=0
MOVL C00944 V=800.0 PL=0
MOVL C00945 V=800.0 PL=0
MOVL C00946 V=800.0 PL=0
MOVL C00947 V=800.0 PL=0
MOVL C00948 V=800.0 PL=0
MOVL C00949 V=800.0 PL=0
MOVL C00950 V=800.0 PL=0
MOVL C00951 V=800.0 PL=0
MOVL C00952 V=800.0 PL=0
MOVL C00953 V=800.0 PL=0
MOVL C00954 V=800.0 PL=0
MOVL C00955 V=800.0 PL=0
MOVL C00956 V=800.0 PL=0
MOVL C00957 V=800.0 PL=0
MOVL C00958 V=800.0 PL=0
MOVL C00959 V=800.0 PL=0
MOVL C00960 V=800.0 PL=0
MOVL C00961 V=800.0 PL=0
MOVL C00962 V=800.0 PL=0
MOVL C00963 V=800.0 PL=0
MOVL C00964 V=800.0 PL=0
MOVL C00965 V=800.0 PL=0
MOVL C00966 V=800.0 PL=0
MOVL C00967 V=800.0 PL=0
MOVL C00968 V=800.0 PL=0
MOVL C00969 V=800.0 PL=0
MOVL C00970 V=800.0 PL=0
MOVL C00971 V=800.0 PL=0
MOVL C00972 V=800.0 PL=0
MOVL C00973 V=800.0 PL=0
MOVL C00974 V=800.0 PL=0
MOVL C00975 V=800.0 PL=0
MOVL C00976 V=800.0 PL=0
MOVL C00977 V=800.0 PL=0
MOVL C00978 V=800.0 PL=0
MOVL C00979 V=800.0 PL=0
MOVL C00980 V=800.0 PL=0
MOVL C00981 V=800.0 PL=0
MOVL C00982 V=800.0 PL=0
MOVL C00983 V=800.0 PL=0
MOVL C00984 V=800.0 PL=0
MOVL C00985 V=800.0 PL=0
MOVL C00986 V=800.0 PL=0
MOVL C00987 V=800.0 PL=0
MOVL C00988 V=800.0 PL=0
MOVL C00989 V=800.0 PL=0
MOVL C00990 V=800.0 PL=0
MOVL C00991 V=800.0 PL=0
MOVL C00992 V=800.0 PL=0
MOVL C00993 V=800.0 PL=0
MOVL C00994 V=800.0 PL=0
MOVL C00995 V=800.0 PL=0
MOVL C00996 V=800.0 PL=0
MOVL C00997 V=800.0 PL=0
MOVL C00998 V=800.0 PL=0
MOVL C00999 V=800.0 PL=0
MOVL C01000 V=800.0 PL=0
MOVL C01001 V=800.0 PL=0
MOVL C01002 V=800.0 PL=0
MOVL C01003 V=800.0 PL=0
MOVL C01004 V=800.0 PL=0
MOVL C01005 V=800.0 PL=0
MOVL C01006 V=800.0 PL=0
MOVL C01007 V=800.0 PL=0
MOVL C01008 V=800.0 PL=0
MOVL C01009 V=800.0 PL=0
MOVL C01010 V=800.0 PL=0
MOVL C01011 V=800.0 PL=0
MOVL C01012 V=800.0 PL=0
MOVL C01013 V=800.0 PL=0
MOVL C01014 V=800.0 PL=0
MOVL C01015 V=800.0 PL=0
MOVL C01016 V=800.0 PL=0
MOVL C01017 V=800.0 PL=0
MOVL C01018 V=800.0 PL=0
MOVL C01019 V=800.0 PL=0
MOVL C01020 V=800.0 PL=0
MOVL C01021 V=800.0 PL=0
MOVL C01022 V=800.0 PL=0
MOVL C01023 V=800.0 PL=0
MOVL C01024 V=800.0 PL=0
MOVL C01025 V=800.0 PL=0
MOVL C01026 V=800.0 PL=0
MOVL C01027 V=800.0 PL=0
MOVL C01028 V=800.0 PL=0
MOVL C01029 V=800.0 PL=0
MOVL C01030 V=800.0 PL=0
MOVL C01031 V=800.0 PL=0
MOVL C01032 V=800.0 PL=0
MOVL C01033 V=800.0 PL=0
MOVL C01034 V=800.0 PL=0
MOVL C01035 V=800.0 PL=0
MOVL C01036 V=800.0 PL=0
MOVL C01037 V=800.0 PL=0
MOVL C01038 V=800.0 PL=0
MOVL C01039 V=800.0 PL=0
MOVL C01040 V=800.0 PL=0
MOVL C01041 V=800.0 PL=0
MOVL C01042 V=800.0 PL=0
MOVL C01043 V=800.0 PL=0
MOVL C01044 V=800.0 PL=0
MOVL C01045 V=800.0 PL=0
MOVL C01046 V=800.0 PL=0
MOVL C01047 V=800.0 PL=0
MOVL C01048 V=800.0 PL=0
MOVL C01049 V=800.0 PL=0
MOVL C01050 V=800.0 PL=0
MOVL C01051 V=800.0 PL=0
MOVL C01052 V=800.0 PL=0
MOVL C01053 V=800.0 PL=0
MOVL C01054 V=800.0 PL=0
MOVL C01055 V=800.0 PL=0
MOVL C01056 V=800.0 PL=0
MOVL C01057 V=800.0 PL=0
MOVL C01058 V=800.0 PL=0
MOVL C01059 V=800.0 PL=0
MOVL C01060 V=800.0 PL=0
MOVL C01061 V=800.0 PL=0
MOVL C01062 V=800.0 PL=0
MOVL C01063 V=800.0 PL=0
MOVL C01064 V=800.0 PL=0
MOVL C01065 V=800.0 PL=0
MOVL C01066 V=800.0 PL=0
MOVL C01067 V=800.0 PL=0
MOVL C01068 V=800.0 PL=0
MOVL C01069 V=800.0 PL=0
MOVL C01070 V=800.0 PL=0
MOVL C01071 V=800.0 PL=0
MOVL C01072 V=800.0 PL=0
MOVL C01073 V=800.0 PL=0
MOVL C01074 V=800.0 PL=0
MOVL C01075 V=800.0 PL=0
MOVL C01076 V=800.0 PL=0
MOVL C01077 V=800.0 PL=0
MOVL C01078 V=800.0 PL=0
MOVL C01079 V=800.0 PL=0
MOVL C01080 V=800.0 PL=0
MOVL C01081 V=800.0 PL=0
MOVL C01082 V=800.0 PL=0
MOVL C01083 V=800.0 PL=0
MOVL C01084 V=800.0 PL=0
MOVL C01085 V=800.0 PL=0
MOVL C01086 V=800.0 PL=0
MOVL C01087 V=800.0 PL=0
MOVL C01088 V=800.0 PL=0
MOVL C01089 V=800.0 PL=0
MOVL C01090 V=800.0 PL=0
MOVL C01091 V=800.0 PL=0
MOVL C01092 V=800.0 PL=0
MOVL C01093 V=800.0 PL=0
MOVL C01094 V=800.0 PL=0
MOVL C01095 V=800.0 PL=0
MOVL C01096 V=800.0 PL=0
MOVL C01097 V=800.0 PL=0
MOVL C01098 V=800.0 PL=0
MOVL C01099 V=800.0 PL=0
MOVL C01100 V=800.0 PL=0
MOVL C01101 V=800.0 PL=0
MOVL C01102 V=800.0 PL=0
MOVL C01103 V=800.0 PL=0
MOVL C01104 V=800.0 PL=0
MOVL C01105 V=800.0 PL=0
MOVL C01106 V=800.0 PL=0
MOVL C01107 V=800.0 PL=0
MOVL C01108 V=800.0 PL=0
MOVL C01109 V=800.0 PL=0
MOVL C01110 V=800.0 PL=0
MOVL C01111 V=800.0 PL=0
MOVL C01112 V=800.0 PL=0
MOVL C01113 V=800.0 PL=0
MOVL C01114 V=800.0 PL=0
MOVL C01115 V=800.0 PL=0
MOVL C01116 V=800.0 PL=0
MOVL C01117 V=800.0 PL=0
MOVL C01118 V=800.0 PL=0
MOVL C01119 V=800.0 PL=0
MOVL C01120 V=800.0 PL=0
MOVL C01121 V=800.0 PL=0
MOVL C01122 V=800.0 PL=0
MOVL C01123 V=800.0 PL=0
MOVL C01124 V=800.0 PL=0
MOVL C01125 V=800.0 PL=0
MOVL C01126 V=800.0 PL=0
MOVL C01127 V=800.0 PL=0
MOVL C01128 V=800.0 PL=0
MOVL C01129 V=800.0 PL=0
MOVL C01130 V=800.0 PL=0
MOVL C01131 V=800.0 PL=0
MOVL C01132 V=800.0 PL=0
MOVL C01133 V=800.0 PL=0
MOVL C01134 V=800.0 PL=0
MOVL C01135 V=800.0 PL=0
MOVL C01136 V=800.0 PL=0
MOVL C01137 V=800.0 PL=0
MOVL C01138 V=800.0 PL=0
MOVL C01139 V=800.0 PL=0
MOVL C01140 V=800.0 PL=0
MOVL C01141 V=800.0 PL=0
MOVL C01142 V=800.0 PL=0
MOVL C01143 V=800.0 PL=0
MOVL C01144 V=800.0 PL=0
MOVL C01145 V=800.0 PL=0
MOVL C01146 V=800.0 PL=0
MOVL C01147 V=800.0 PL=0
MOVL C01148 V=800.0 PL=0
MOVL C01149 V=800.0 PL=0
MOVL C01150 V=800.0 PL=0
MOVL C01151 V=800.0 PL=0
MOVL C01152 V=800.0 PL=0
MOVL C01153 V=800.0 PL=0
MOVL C01154 V=800.0 PL=0
MOVL C01155 V=800.0 PL=0
MOVL C01156 V=800.0 PL=0
MOVL C01157 V=800.0 PL=0
MOVL C01158 V=800.0 PL=0
MOVL C01159 V=800.0 PL=0
MOVL C01160 V=800.0 PL=0
MOVL C01161 V=800.0 PL=0
MOVL C01162 V=800.0 PL=0
MOVL C01163 V=800.0 PL=0
MOVL C01164 V=800.0 PL=0
MOVL C01165 V=800.0 PL=0
MOVL C01166 V=800.0 PL=0
MOVL C01167 V=800.0 PL=0
MOVL C01168 V=800.0 PL=0
MOVL C01169 V=800.0 PL=0
MOVL C01170 V=800.0 PL=0
MOVL C01171 V=800.0 PL=0
MOVL C01172 V=800.0 PL=0
MOVL C01173 V=800.0 PL=0
MOVL C01174 V=800.0 PL=0
MOVL C01175 V=800.0 PL=0
MOVL C01176 V=800.0 PL=0
MOVL C01177 V=800.0 PL=0
MOVL C01178 V=800.0 PL=0
MOVL C01179 V=800.0 PL=0
MOVL C01180 V=800.0 PL=0
MOVL C01181 V=800.0 PL=0
MOVL C01182 V=800.0 PL=0
MOVL C01183 V=800.0 PL=0
MOVL C01184 V=800.0 PL=0
MOVL C01185 V=800.0 PL=0
MOVL C01186 V=800.0 PL=0
MOVL C01187 V=800.0 PL=0
MOVL C01188 V=800.0 PL=0
MOVL C01189 V=800.0 PL=0
MOVL C01190 V=800.0 PL=0
MOVL C01191 V=800.0 PL=0
MOVL C01192 V=800.0 PL=0
MOVL C01193 V=800.0 PL=0
MOVL C01194 V=800.0 PL=0
MOVL C01195 V=800.0 PL=0
MOVL C01196 V=800.0 PL=0
MOVL C01197 V=800.0 PL=0
MOVL C01198 V=800.0 PL=0
MOVL C01199 V=800.0 PL=0
MOVL C01200 V=800.0 PL=0
MOVL C01201 V=800.0 PL=0
MOVL C01202 V=800.0 PL=0
MOVL C01203 V=800.0 PL=0
MOVL C01204 V=800.0 PL=0
MOVL C01205 V=800.0 PL=0
MOVL C01206 V=800.0 PL=0
MOVL C01207 V=800.0 PL=0
MOVL C01208 V=800.0 PL=0
MOVL C01209 V=800.0 PL=0
MOVL C01210 V=800.0 PL=0
MOVL C01211 V=800.0 PL=0
MOVL C01212 V=800.0 PL=0
MOVL C01213 V=800.0 PL=0
MOVL C01214 V=800.0 PL=0
MOVL C01215 V=800.0 PL=0
MOVL C01216 V=800.0 PL=0
MOVL C01217 V=800.0 PL=0
MOVL C01218 V=800.0 PL=0
MOVL C01219 V=800.0 PL=0
MOVL C01220 V=800.0 PL=0
MOVL C01221 V=800.0 PL=0
MOVL C01222 V=800.0 PL=0
MOVL C01223 V=800.0 PL=0
MOVL C01224 V=800.0 PL=0
MOVL C01225 V=800.0 PL=0
MOVL C01226 V=800.0 PL=0
MOVL C01227 V=800.0 PL=0
MOVL C01228 V=800.0 PL=0
MOVL C01229 V=800.0 PL=0
MOVL C01230 V=800.0 PL=0
MOVL C01231 V=800.0 PL=0
MOVL C01232 V=800.0 PL=0
MOVL C01233 V=800.0 PL=0
MOVL C01234 V=800.0 PL=0
MOVL C01235 V=800.0 PL=0
MOVL C01236 V=800.0 PL=0
MOVL C01237 V=800.0 PL=0
MOVL C01238 V=800.0 PL=0
MOVL C01239 V=800.0 PL=0
MOVL C01240 V=800.0 PL=0
MOVL C01241 V=800.0 PL=0
MOVL C01242 V=800.0 PL=0
MOVL C01243 V=800.0 PL=0
MOVL C01244 V=800.0 PL=0
MOVL C01245 V=800.0 PL=0
MOVL C01246 V=800.0 PL=0
MOVL C01247 V=800.0 PL=0
MOVL C01248 V=800.0 PL=0
MOVL C01249 V=800.0 PL=0
MOVL C01250 V=800.0 PL=0
MOVL C01251 V=800.0 PL=0
MOVL C01252 V=800.0 PL=0
MOVL C01253 V=800.0 PL=0
MOVL C01254 V=800.0 PL=0
MOVL C01255 V=800.0 PL=0
MOVL C01256 V=800.0 PL=0
MOVL C01257 V=800.0 PL=0
MOVL C01258 V=800.0 PL=0
MOVL C01259 V=800.0 PL=0
MOVL C01260 V=800.0 PL=0
MOVL C01261 V=800.0 PL=0
MOVL C01262 V=800.0 PL=0
MOVL C01263 V=800.0 PL=0
MOVL C01264 V=800.0 PL=0
MOVL C01265 V=800.0 PL=0
MOVL C01266 V=800.0 PL=0
MOVL C01267 V=800.0 PL=0
MOVL C01268 V=800.0 PL=0
MOVL C01269 V=800.0 PL=0
MOVL C01270 V=800.0 PL=0
MOVL C01271 V=800.0 PL=0
MOVL C01272 V=800.0 PL=0
MOVL C01273 V=800.0 PL=0
MOVL C01274 V=800.0 PL=0
MOVL C01275 V=800.0 PL=0
MOVL C01276 V=800.0 PL=0
MOVL C01277 V=800.0 PL=0
MOVL C01278 V=800.0 PL=0
MOVL C01279 V=800.0 PL=0
MOVL C01280 V=800.0 PL=0
MOVL C01281 V=800.0 PL=0
MOVL C01282 V=800.0 PL=0
MOVL C01283 V=800.0 PL=0
MOVL C01284 V=800.0 PL=0
MOVL C01285 V=800.0 PL=0
MOVL C01286 V=800.0 PL=0
MOVL C01287 V=800.0 PL=0
MOVL C01288 V=800.0 PL=0
MOVL C01289 V=800.0 PL=0
MOVL C01290 V=800.0 PL=0
MOVL C01291 V=800.0 PL=0
MOVL C01292 V=800.0 PL=0
MOVL C01293 V=800.0 PL=0
MOVL C01294 V=800.0 PL=0
MOVL C01295 V=800.0 PL=0
MOVL C01296 V=800.0 PL=0
MOVL C01297 V=800.0 PL=0
MOVL C01298 V=800.0 PL=0
MOVL C01299 V=800.0 PL=0
MOVL C01300 V=800.0 PL=0
MOVL C01301 V=800.0 PL=0
MOVL C01302 V=800.0 PL=0
MOVL C01303 V=800.0 PL=0
MOVL C01304 V=800.0 PL=0
MOVL C01305 V=800.0 PL=0
MOVL C01306 V=800.0 PL=0
MOVL C01307 V=800.0 PL=0
MOVL C01308 V=800.0 PL=0
MOVL C01309 V=800.0 PL=0
MOVL C01310 V=800.0 PL=0
MOVL C01311 V=800.0 PL=0
MOVL C01312 V=800.0 PL=0
MOVL C01313 V=800.0 PL=0
MOVL C01314 V=800.0 PL=0
MOVL C01315 V=800.0 PL=0
MOVL C01316 V=800.0 PL=0
MOVL C01317 V=800.0 PL=0
MOVL C01318 V=800.0 PL=0
MOVL C01319 V=800.0 PL=0
MOVL C01320 V=800.0 PL=0
MOVL C01321 V=800.0 PL=0
MOVL C01322 V=800.0 PL=0
MOVL C01323 V=800.0 PL=0
MOVL C01324 V=800.0 PL=0
MOVL C01325 V=800.0 PL=0
MOVL C01326 V=800.0 PL=0
MOVL C01327 V=800.0 PL=0
MOVL C01328 V=800.0 PL=0
MOVL C01329 V=800.0 PL=0
MOVL C01330 V=800.0 PL=0
MOVL C01331 V=800.0 PL=0
MOVL C01332 V=800.0 PL=0
MOVL C01333 V=800.0 PL=0
MOVL C01334 V=800.0 PL=0
MOVL C01335 V=800.0 PL=0
MOVL C01336 V=800.0 PL=0
MOVL C01337 V=800.0 PL=0
MOVL C01338 V=800.0 PL=0
MOVL C01339 V=800.0 PL=0
MOVL C01340 V=800.0 PL=0
MOVL C01341 V=800.0 PL=0
MOVL C01342 V=800.0 PL=0
MOVL C01343 V=800.0 PL=0
MOVL C01344 V=800.0 PL=0
MOVL C01345 V=800.0 PL=0
MOVL C01346 V=800.0 PL=0
MOVL C01347 V=800.0 PL=0
MOVL C01348 V=800.0 PL=0
MOVL C01349 V=800.0 PL=0
MOVL C01350 V=800.0 PL=0
MOVL C01351 V=800.0 PL=0
MOVL C01352 V=800.0 PL=0
MOVL C01353 V=800.0 PL=0
MOVL C01354 V=800.0 PL=0
MOVL C01355 V=800.0 PL=0
MOVL C01356 V=800.0 PL=0
MOVL C01357 V=800.0 PL=0
MOVL C01358 V=800.0 PL=0
MOVL C01359 V=800.0 PL=0
MOVL C01360 V=800.0 PL=0
MOVL C01361 V=800.0 PL=0
MOVL C01362 V=800.0 PL=0
MOVL C01363 V=800.0 PL=0
MOVL C01364 V=800.0 PL=0
MOVL C01365 V=800.0 PL=0
MOVL C01366 V=800.0 PL=0
MOVL C01367 V=800.0 PL=0
MOVL C01368 V=800.0 PL=0
MOVL C01369 V=800.0 PL=0
MOVL C01370 V=800.0 PL=0
MOVL C01371 V=800.0 PL=0
MOVL C01372 V=800.0 PL=0
MOVL C01373 V=800.0 PL=0
MOVL C01374 V=800.0 PL=0
MOVL C01375 V=800.0 PL=0
MOVL C01376 V=800.0 PL=0
MOVL C01377 V=800.0 PL=0
MOVL C01378 V=800.0 PL=0
MOVL C01379 V=800.0 PL=0
MOVL C01380 V=800.0 PL=0
MOVL C01381 V=800.0 PL=0
MOVL C01382 V=800.0 PL=0
MOVL C01383 V=800.0 PL=0
MOVL C01384 V=800.0 PL=0
MOVL C01385 V=800.0 PL=0
MOVL C01386 V=800.0 PL=0
MOVL C01387 V=800.0 PL=0
MOVL C01388 V=800.0 PL=0
MOVL C01389 V=800.0 PL=0
MOVL C01390 V=800.0 PL=0
MOVL C01391 V=800.0 PL=0
MOVL C01392 V=800.0 PL=0
MOVL C01393 V=800.0 PL=0
MOVL C01394 V=800.0 PL=0
MOVL C01395 V=800.0 PL=0
MOVL C01396 V=800.0 PL=0
MOVL C01397 V=800.0 PL=0
MOVL C01398 V=800.0 PL=0
MOVL C01399 V=800.0 PL=0
MOVL C01400 V=800.0 PL=0
MOVL C01401 V=800.0 PL=0
MOVL C01402 V=800.0 PL=0
MOVL C01403 V=800.0 PL=0
MOVL C01404 V=800.0 PL=0
MOVL C01405 V=800.0 PL=0
MOVL C01406 V=800.0 PL=0
MOVL C01407 V=800.0 PL=0
MOVL C01408 V=800.0 PL=0
MOVL C01409 V=800.0 PL=0
MOVL C01410 V=800.0 PL=0
MOVL C01411 V=800.0 PL=0
MOVL C01412 V=800.0 PL=0
MOVL C01413 V=800.0 PL=0
MOVL C01414 V=800.0 PL=0
MOVL C01415 V=800.0 PL=0
MOVL C01416 V=800.0 PL=0
MOVL C01417 V=800.0 PL=0
MOVL C01418 V=800.0 PL=0
MOVL C01419 V=800.0 PL=0
MOVL C01420 V=800.0 PL=0
MOVL C01421 V=800.0 PL=0
MOVL C01422 V=800.0 PL=0
MOVL C01423 V=800.0 PL=0
MOVL C01424 V=800.0 PL=0
MOVL C01425 V=800.0 PL=0
MOVL C01426 V=800.0 PL=0
MOVL C01427 V=800.0 PL=0
MOVL C01428 V=800.0 PL=0
MOVL C01429 V=800.0 PL=0
MOVL C01430 V=800.0 PL=0
MOVL C01431 V=800.0 PL=0
MOVL C01432 V=800.0 PL=0
MOVL C01433 V=800.0 PL=0
MOVL C01434 V=800.0 PL=0
MOVL C01435 V=800.0 PL=0
MOVL C01436 V=800.0 PL=0
MOVL C01437 V=800.0 PL=0
MOVL C01438 V=800.0 PL=0
MOVL C01439 V=800.0 PL=0
MOVL C01440 V=800.0 PL=0
MOVL C01441 V=800.0 PL=0
MOVL C01442 V=800.0 PL=0
MOVL C01443 V=800.0 PL=0
MOVL C01444 V=800.0 PL=0
MOVL C01445 V=800.0 PL=0
MOVL C01446 V=800.0 PL=0
MOVL C01447 V=800.0 PL=0
MOVL C01448 V=800.0 PL=0
MOVL C01449 V=800.0 PL=0
MOVL C01450 V=800.0 PL=0
MOVL C01451 V=800.0 PL=0
MOVL C01452 V=800.0 PL=0
MOVL C01453 V=800.0 PL=0
MOVL C01454 V=800.0 PL=0
MOVL C01455 V=800.0 PL=0
MOVL C01456 V=800.0 PL=0
MOVL C01457 V=800.0 PL=0
MOVL C01458 V=800.0 PL=0
MOVL C01459 V=800.0 PL=0
MOVL C01460 V=800.0 PL=0
MOVL C01461 V=800.0 PL=0
MOVL C01462 V=800.0 PL=0
MOVL C01463 V=800.0 PL=0
MOVL C01464 V=800.0 PL=0
MOVL C01465 V=800.0 PL=0
MOVL C01466 V=800.0 PL=0
MOVL C01467 V=800.0 PL=0
MOVL C01468 V=800.0 PL=0
MOVL C01469 V=800.0 PL=0
MOVL C01470 V=800.0 PL=0
MOVL C01471 V=800.0 PL=0
MOVL C01472 V=800.0 PL=0
MOVL C01473 V=800.0 PL=0
MOVL C01474 V=800.0 PL=0
MOVL C01475 V=800.0 PL=0
MOVL C01476 V=800.0 PL=0
MOVL C01477 V=800.0 PL=0
MOVL C01478 V=800.0 PL=0
MOVL C01479 V=800.0 PL=0
MOVL C01480 V=800.0 PL=0
MOVL C01481 V=800.0 PL=0
MOVL C01482 V=800.0 PL=0
MOVL C01483 V=800.0 PL=0
MOVL C01484 V=800.0 PL=0
MOVL C01485 V=800.0 PL=0
MOVL C01486 V=800.0 PL=0
MOVL C01487 V=800.0 PL=0
MOVL C01488 V=800.0 PL=0
MOVL C01489 V=800.0 PL=0
MOVL C01490 V=800.0 PL=0
MOVL C01491 V=800.0 PL=0
MOVL C01492 V=800.0 PL=0
MOVL C01493 V=800.0 PL=0
MOVL C01494 V=800.0 PL=0
MOVL C01495 V=800.0 PL=0
MOVL C01496 V=800.0 PL=0
MOVL C01497 V=800.0 PL=0
MOVL C01498 V=800.0 PL=0
MOVL C01499 V=800.0 PL=0
MOVL C01500 V=800.0 PL=0
MOVL C01501 V=800.0 PL=0
MOVL C01502 V=800.0 PL=0
MOVL C01503 V=800.0 PL=0
MOVL C01504 V=800.0 PL=0
MOVL C01505 V=800.0 PL=0
MOVL C01506 V=800.0 PL=0
MOVL C01507 V=800.0 PL=0
MOVL C01508 V=800.0 PL=0
MOVL C01509 V=800.0 PL=0
MOVL C01510 V=800.0 PL=0
MOVL C01511 V=800.0 PL=0
MOVL C01512 V=800.0 PL=0
MOVL C01513 V=800.0 PL=0
MOVL C01514 V=800.0 PL=0
MOVL C01515 V=800.0 PL=0
MOVL C01516 V=800.0 PL=0
MOVL C01517 V=800.0 PL=0
MOVL C01518 V=800.0 PL=0
MOVL C01519 V=800.0 PL=0
MOVL C01520 V=800.0 PL=0
MOVL C01521 V=800.0 PL=0
MOVL C01522 V=800.0 PL=0
MOVL C01523 V=800.0 PL=0
MOVL C01524 V=800.0 PL=0
MOVL C01525 V=800.0 PL=0
MOVL C01526 V=800.0 PL=0
MOVL C01527 V=800.0 PL=0
MOVL C01528 V=800.0 PL=0
MOVL C01529 V=800.0 PL=0
MOVL C01530 V=800.0 PL=0
MOVL C01531 V=800.0 PL=0
MOVL C01532 V=800.0 PL=0
MOVL C01533 V=800.0 PL=0
MOVL C01534 V=800.0 PL=0
MOVL C01535 V=800.0 PL=0
MOVL C01536 V=800.0 PL=0
MOVL C01537 V=800.0 PL=0
MOVL C01538 V=800.0 PL=0
MOVL C01539 V=800.0 PL=0
MOVL C01540 V=800.0 PL=0
MOVL C01541 V=800.0 PL=0
MOVL C01542 V=800.0 PL=0
MOVL C01543 V=800.0 PL=0
MOVL C01544 V=800.0 PL=0
MOVL C01545 V=800.0 PL=0
MOVL C01546 V=800.0 PL=0
MOVL C01547 V=800.0 PL=0
MOVL C01548 V=800.0 PL=0
MOVL C01549 V=800.0 PL=0
MOVL C01550 V=800.0 PL=0
MOVL C01551 V=800.0 PL=0
MOVL C01552 V=800.0 PL=0
MOVL C01553 V=800.0 PL=0
MOVL C01554 V=800.0 PL=0
MOVL C01555 V=800.0 PL=0
MOVL C01556 V=800.0 PL=0
MOVL C01557 V=800.0 PL=0
MOVL C01558 V=800.0 PL=0
MOVL C01559 V=800.0 PL=0
MOVL C01560 V=800.0 PL=0
MOVL C01561 V=800.0 PL=0
MOVL C01562 V=800.0 PL=0
MOVL C01563 V=800.0 PL=0
MOVL C01564 V=800.0 PL=0
MOVL C01565 V=800.0 PL=0
MOVL C01566 V=800.0 PL=0
MOVL C01567 V=800.0 PL=0
MOVL C01568 V=800.0 PL=0
MOVL C01569 V=800.0 PL=0
MOVL C01570 V=800.0 PL=0
MOVL C01571 V=800.0 PL=0
MOVL C01572 V=800.0 PL=0
MOVL C01573 V=800.0 PL=0
MOVL C01574 V=800.0 PL=0
MOVL C01575 V=800.0 PL=0
MOVL C01576 V=800.0 PL=0
MOVL C01577 V=800.0 PL=0
MOVL C01578 V=800.0 PL=0
MOVL C01579 V=800.0 PL=0
MOVL C01580 V=800.0 PL=0
MOVL C01581 V=800.0 PL=0
MOVL C01582 V=800.0 PL=0
MOVL C01583 V=800.0 PL=0
MOVL C01584 V=800.0 PL=0
MOVL C01585 V=800.0 PL=0
MOVL C01586 V=800.0 PL=0
MOVL C01587 V=800.0 PL=0
MOVL C01588 V=800.0 PL=0
MOVL C01589 V=800.0 PL=0
MOVL C01590 V=800.0 PL=0
MOVL C01591 V=800.0 PL=0
MOVL C01592 V=800.0 PL=0
MOVL C01593 V=800.0 PL=0
MOVL C01594 V=800.0 PL=0
MOVL C01595 V=800.0 PL=0
MOVL C01596 V=800.0 PL=0
MOVL C01597 V=800.0 PL=0
MOVL C01598 V=800.0 PL=0
MOVL C01599 V=800.0 PL=0
MOVL C01600 V=800.0 PL=0
MOVL C01601 V=800.0 PL=0
MOVL C01602 V=800.0 PL=0
MOVL C01603 V=800.0 PL=0
MOVL C01604 V=800.0 PL=0
MOVL C01605 V=800.0 PL=0
MOVL C01606 V=800.0 PL=0
MOVL C01607 V=800.0 PL=0
MOVL C01608 V=800.0 PL=0
MOVL C01609 V=800.0 PL=0
MOVL C01610 V=800.0 PL=0
MOVL C01611 V=800.0 PL=0
MOVL C01612 V=800.0 PL=0
MOVL C01613 V=800.0 PL=0
MOVL C01614 V=800.0 PL=0
MOVL C01615 V=800.0 PL=0
MOVL C01616 V=800.0 PL=0
MOVL C01617 V=800.0 PL=0
MOVL C01618 V=800.0 PL=0
MOVL C01619 V=800.0 PL=0
MOVL C01620 V=800.0 PL=0
MOVL C01621 V=800.0 PL=0
MOVL C01622 V=800.0 PL=0
MOVL C01623 V=800.0 PL=0
MOVL C01624 V=800.0 PL=0
MOVL C01625 V=800.0 PL=0
MOVL C01626 V=800.0 PL=0
MOVL C01627 V=800.0 PL=0
MOVL C01628 V=800.0 PL=0
MOVL C01629 V=800.0 PL=0
MOVL C01630 V=800.0 PL=0
MOVL C01631 V=800.0 PL=0
MOVL C01632 V=800.0 PL=0
MOVL C01633 V=800.0 PL=0
MOVL C01634 V=800.0 PL=0
MOVL C01635 V=800.0 PL=0
MOVL C01636 V=800.0 PL=0
MOVL C01637 V=800.0 PL=0
MOVL C01638 V=800.0 PL=0
MOVL C01639 V=800.0 PL=0
MOVL C01640 V=800.0 PL=0
MOVL C01641 V=800.0 PL=0
MOVL C01642 V=800.0 PL=0
MOVL C01643 V=800.0 PL=0
MOVL C01644 V=800.0 PL=0
MOVL C01645 V=800.0 PL=0
MOVL C01646 V=800.0 PL=0
MOVL C01647 V=800.0 PL=0
MOVL C01648 V=800.0 PL=0
MOVL C01649 V=800.0 PL=0
MOVL C01650 V=800.0 PL=0
MOVL C01651 V=800.0 PL=0
MOVL C01652 V=800.0 PL=0
MOVL C01653 V=800.0 PL=0
MOVL C01654 V=800.0 PL=0
MOVL C01655 V=800.0 PL=0
MOVL C01656 V=800.0 PL=0
MOVL C01657 V=800.0 PL=0
MOVL C01658 V=800.0 PL=0
MOVL C01659 V=800.0 PL=0
MOVL C01660 V=800.0 PL=0
MOVL C01661 V=800.0 PL=0
MOVL C01662 V=800.0 PL=0
MOVL C01663 V=800.0 PL=0
MOVL C01664 V=800.0 PL=0
MOVL C01665 V=800.0 PL=0
MOVL C01666 V=800.0 PL=0
MOVL C01667 V=800.0 PL=0
MOVL C01668 V=800.0 PL=0
MOVL C01669 V=800.0 PL=0
MOVL C01670 V=800.0 PL=0
MOVL C01671 V=800.0 PL=0
MOVL C01672 V=800.0 PL=0
MOVL C01673 V=800.0 PL=0
MOVL C01674 V=800.0 PL=0
MOVL C01675 V=800.0 PL=0
MOVL C01676 V=800.0 PL=0
MOVL C01677 V=800.0 PL=0
MOVL C01678 V=800.0 PL=0
MOVL C01679 V=800.0 PL=0
MOVL C01680 V=800.0 PL=0
MOVL C01681 V=800.0 PL=0
MOVL C01682 V=800.0 PL=0
MOVL C01683 V=800.0 PL=0
MOVL C01684 V=800.0 PL=0
MOVL C01685 V=800.0 PL=0
MOVL C01686 V=800.0 PL=0
MOVL C01687 V=800.0 PL=0
MOVL C01688 V=800.0 PL=0
MOVL C01689 V=800.0 PL=0
MOVL C01690 V=800.0 PL=0
MOVL C01691 V=800.0 PL=0
MOVL C01692 V=800.0 PL=0
MOVL C01693 V=800.0 PL=0
MOVL C01694 V=800.0 PL=0
MOVL C01695 V=800.0 PL=0
MOVL C01696 V=800.0 PL=0
MOVL C01697 V=800.0 PL=0
MOVL C01698 V=800.0 PL=0
MOVL C01699 V=800.0 PL=0
MOVL C01700 V=800.0 PL=0
MOVL C01701 V=800.0 PL=0
MOVL C01702 V=800.0 PL=0
MOVL C01703 V=800.0 PL=0
MOVL C01704 V=800.0 PL=0
MOVL C01705 V=800.0 PL=0
MOVL C01706 V=800.0 PL=0
MOVL C01707 V=800.0 PL=0
MOVL C01708 V=800.0 PL=0
MOVL C01709 V=800.0 PL=0
MOVL C01710 V=800.0 PL=0
MOVL C01711 V=800.0 PL=0
MOVL C01712 V=800.0 PL=0
MOVL C01713 V=800.0 PL=0
MOVL C01714 V=800.0 PL=0
MOVL C01715 V=800.0 PL=0
MOVL C01716 V=800.0 PL=0
MOVL C01717 V=800.0 PL=0
MOVL C01718 V=800.0 PL=0
MOVL C01719 V=800.0 PL=0
MOVL C01720 V=800.0 PL=0
MOVL C01721 V=800.0 PL=0
MOVL C01722 V=800.0 PL=0
MOVL C01723 V=800.0 PL=0
MOVL C01724 V=800.0 PL=0
MOVL C01725 V=800.0 PL=0
MOVL C01726 V=800.0 PL=0
MOVL C01727 V=800.0 PL=0
MOVL C01728 V=800.0 PL=0
MOVL C01729 V=800.0 PL=0
MOVL C01730 V=800.0 PL=0
MOVL C01731 V=800.0 PL=0
MOVL C01732 V=800.0 PL=0
MOVL C01733 V=800.0 PL=0
MOVL C01734 V=800.0 PL=0
MOVL C01735 V=800.0 PL=0
MOVL C01736 V=800.0 PL=0
MOVL C01737 V=800.0 PL=0
MOVL C01738 V=800.0 PL=0
MOVL C01739 V=800.0 PL=0
MOVL C01740 V=800.0 PL=0
MOVL C01741 V=800.0 PL=0
MOVL C01742 V=800.0 PL=0
MOVL C01743 V=800.0 PL=0
MOVL C01744 V=800.0 PL=0
MOVL C01745 V=800.0 PL=0
MOVL C01746 V=800.0 PL=0
MOVL C01747 V=800.0 PL=0
MOVL C01748 V=800.0 PL=0
MOVL C01749 V=800.0 PL=0
MOVL C01750 V=800.0 PL=0
MOVL C01751 V=800.0 PL=0
MOVL C01752 V=800.0 PL=0
MOVL C01753 V=800.0 PL=0
MOVL C01754 V=800.0 PL=0
MOVL C01755 V=800.0 PL=0
MOVL C01756 V=800.0 PL=0
MOVL C01757 V=800.0 PL=0
MOVL C01758 V=800.0 PL=0
MOVL C01759 V=800.0 PL=0
MOVL C01760 V=800.0 PL=0
MOVL C01761 V=800.0 PL=0
MOVL C01762 V=800.0 PL=0
MOVL C01763 V=800.0 PL=0
MOVL C01764 V=800.0 PL=0
MOVL C01765 V=800.0 PL=0
MOVL C01766 V=800.0 PL=0
MOVL C01767 V=800.0 PL=0
MOVL C01768 V=800.0 PL=0
MOVL C01769 V=800.0 PL=0
MOVL C01770 V=800.0 PL=0
MOVL C01771 V=800.0 PL=0
MOVL C01772 V=800.0 PL=0
MOVL C01773 V=800.0 PL=0
MOVL C01774 V=800.0 PL=0
MOVL C01775 V=800.0 PL=0
MOVL C01776 V=800.0 PL=0
MOVL C01777 V=800.0 PL=0
MOVL C01778 V=800.0 PL=0
MOVL C01779 V=800.0 PL=0
MOVL C01780 V=800.0 PL=0
MOVL C01781 V=800.0 PL=0
MOVL C01782 V=800.0 PL=0
MOVL C01783 V=800.0 PL=0
MOVL C01784 V=800.0 PL=0
MOVL C01785 V=800.0 PL=0
MOVL C01786 V=800.0 PL=0
MOVL C01787 V=800.0 PL=0
MOVL C01788 V=800.0 PL=0
MOVL C01789 V=800.0 PL=0
MOVL C01790 V=800.0 PL=0
MOVL C01791 V=800.0 PL=0
MOVL C01792 V=800.0 PL=0
MOVL C01793 V=800.0 PL=0
MOVL C01794 V=800.0 PL=0
MOVL C01795 V=800.0 PL=0
MOVL C01796 V=800.0 PL=0
MOVL C01797 V=800.0 PL=0
MOVL C01798 V=800.0 PL=0
MOVL C01799 V=800.0 PL=0
MOVL C01800 V=800.0 PL=0
MOVL C01801 V=800.0 PL=0
MOVL C01802 V=800.0 PL=0
MOVL C01803 V=800.0 PL=0
MOVL C01804 V=800.0 PL=0
MOVL C01805 V=800.0 PL=0
MOVL C01806 V=800.0 PL=0
MOVL C01807 V=800.0 PL=0
MOVL C01808 V=800.0 PL=0
MOVL C01809 V=800.0 PL=0
MOVL C01810 V=800.0 PL=0
MOVL C01811 V=800.0 PL=0
MOVL C01812 V=800.0 PL=0
MOVL C01813 V=800.0 PL=0
MOVL C01814 V=800.0 PL=0
MOVL C01815 V=800.0 PL=0
MOVL C01816 V=800.0 PL=0
MOVL C01817 V=800.0 PL=0
MOVL C01818 V=800.0 PL=0
MOVL C01819 V=800.0 PL=0
MOVL C01820 V=800.0 PL=0
MOVL C01821 V=800.0 PL=0
MOVL C01822 V=800.0 PL=0
MOVL C01823 V=800.0 PL=0
MOVL C01824 V=800.0 PL=0
MOVL C01825 V=800.0 PL=0
MOVL C01826 V=800.0 PL=0
MOVL C01827 V=800.0 PL=0
MOVL C01828 V=800.0 PL=0
MOVL C01829 V=800.0 PL=0
MOVL C01830 V=800.0 PL=0
MOVL C01831 V=800.0 PL=0
MOVL C01832 V=800.0 PL=0
MOVL C01833 V=800.0 PL=0
MOVL C01834 V=800.0 PL=0
MOVL C01835 V=800.0 PL=0
MOVL C01836 V=800.0 PL=0
MOVL C01837 V=800.0 PL=0
MOVL C01838 V=800.0 PL=0
MOVL C01839 V=800.0 PL=0
MOVL C01840 V=800.0 PL=0
MOVL C01841 V=800.0 PL=0
MOVL C01842 V=800.0 PL=0
MOVL C01843 V=800.0 PL=0
MOVL C01844 V=800.0 PL=0
MOVL C01845 V=800.0 PL=0
MOVL C01846 V=800.0 PL=0
MOVL C01847 V=800.0 PL=0
MOVL C01848 V=800.0 PL=0
MOVL C01849 V=800.0 PL=0
MOVL C01850 V=800.0 PL=0
MOVL C01851 V=800.0 PL=0
MOVL C01852 V=800.0 PL=0
MOVL C01853 V=800.0 PL=0
MOVL C01854 V=800.0 PL=0
MOVL C01855 V=800.0 PL=0
MOVL C01856 V=800.0 PL=0
MOVL C01857 V=800.0 PL=0
MOVL C01858 V=800.0 PL=0
MOVL C01859 V=800.0 PL=0
MOVL C01860 V=800.0 PL=0
MOVL C01861 V=800.0 PL=0
MOVL C01862 V=800.0 PL=0
MOVL C01863 V=800.0 PL=0
MOVL C01864 V=800.0 PL=0
MOVL C01865 V=800.0 PL=0
MOVL C01866 V=800.0 PL=0
MOVL C01867 V=800.0 PL=0
MOVL C01868 V=800.0 PL=0
MOVL C01869 V=800.0 PL=0
MOVL C01870 V=800.0 PL=0
MOVL C01871 V=800.0 PL=0
MOVL C01872 V=800.0 PL=0
MOVL C01873 V=800.0 PL=0
MOVL C01874 V=800.0 PL=0
MOVL C01875 V=800.0 PL=0
MOVL C01876 V=800.0 PL=0
MOVL C01877 V=800.0 PL=0
MOVL C01878 V=800.0 PL=0
MOVL C01879 V=800.0 PL=0
MOVL C01880 V=800.0 PL=0
MOVL C01881 V=800.0 PL=0
MOVL C01882 V=800.0 PL=0
MOVL C01883 V=800.0 PL=0
MOVL C01884 V=800.0 PL=0
MOVL C01885 V=800.0 PL=0
MOVL C01886 V=800.0 PL=0
MOVL C01887 V=800.0 PL=0
MOVL C01888 V=800.0 PL=0
MOVL C01889 V=800.0 PL=0
MOVL C01890 V=800.0 PL=0
MOVL C01891 V=800.0 PL=0
MOVL C01892 V=800.0 PL=0
MOVL C01893 V=800.0 PL=0
MOVL C01894 V=800.0 PL=0
MOVL C01895 V=800.0 PL=0
